	VAR jointtarget SDP_1960 := [[-7.34, 34.53, 8.17, 0, 47.31, -84.1], [9E9, 9E9, 9E9, 9E9, 9E9, 9E9]];
	VAR jointtarget SDP_1961 := [[-7.2, 34.54, 8.14, 0, 47.32, -83.96], [9E9, 9E9, 9E9, 9E9, 9E9, 9E9]];
	VAR jointtarget SDP_1962 := [[-7.06, 34.55, 8.12, 0, 47.33, -83.82], [9E9, 9E9, 9E9, 9E9, 9E9, 9E9]];
	VAR jointtarget SDP_1963 := [[-6.92, 34.57, 8.09, 0, 47.34, -83.68], [9E9, 9E9, 9E9, 9E9, 9E9, 9E9]];
	VAR jointtarget SDP_1964 := [[-6.79, 34.58, 8.06, 0, 47.36, -83.55], [9E9, 9E9, 9E9, 9E9, 9E9, 9E9]];
	VAR jointtarget SDP_1965 := [[-6.65, 34.6, 8.03, 0, 47.37, -83.41], [9E9, 9E9, 9E9, 9E9, 9E9, 9E9]];
	VAR jointtarget SDP_1966 := [[-6.51, 34.61, 8, 0, 47.38, -83.27], [9E9, 9E9, 9E9, 9E9, 9E9, 9E9]];
	VAR jointtarget SDP_1967 := [[-6.38, 34.63, 7.97, 0, 47.39, -83.14], [9E9, 9E9, 9E9, 9E9, 9E9, 9E9]];
	VAR jointtarget SDP_1968 := [[-6.24, 34.65, 7.94, 0, 47.41, -83], [9E9, 9E9, 9E9, 9E9, 9E9, 9E9]];
	VAR jointtarget SDP_1969 := [[-6.1, 34.66, 7.91, 0, 47.42, -82.86], [9E9, 9E9, 9E9, 9E9, 9E9, 9E9]];
	VAR jointtarget SDP_1970 := [[-6.07, 34.67, 7.91, 0, 47.43, -83.49], [9E9, 9E9, 9E9, 9E9, 9E9, 9E9]];
	VAR jointtarget SDP_1971 := [[-6.03, 34.67, 7.9, 0, 47.43, -84.78], [9E9, 9E9, 9E9, 9E9, 9E9, 9E9]];
	VAR jointtarget SDP_1972 := [[-6, 34.67, 7.9, 0, 47.43, -86.07], [9E9, 9E9, 9E9, 9E9, 9E9, 9E9]];
	VAR jointtarget SDP_1973 := [[-5.97, 34.67, 7.89, 0, 47.43, -87.36], [9E9, 9E9, 9E9, 9E9, 9E9, 9E9]];
	VAR jointtarget SDP_1974 := [[-5.93, 34.67, 7.89, 0, 47.43, -88.65], [9E9, 9E9, 9E9, 9E9, 9E9, 9E9]];
	VAR jointtarget SDP_1975 := [[-5.9, 34.67, 7.89, 0, 47.43, -89.94], [9E9, 9E9, 9E9, 9E9, 9E9, 9E9]];
	VAR jointtarget SDP_1976 := [[-5.86, 34.67, 7.89, 0, 47.43, -91.23], [9E9, 9E9, 9E9, 9E9, 9E9, 9E9]];
	VAR jointtarget SDP_1977 := [[-5.83, 34.67, 7.9, 0, 47.43, -92.52], [9E9, 9E9, 9E9, 9E9, 9E9, 9E9]];
	VAR jointtarget SDP_1978 := [[-5.79, 34.67, 7.9, 0, 47.43, -93.81], [9E9, 9E9, 9E9, 9E9, 9E9, 9E9]];
	VAR jointtarget SDP_1979 := [[-5.76, 34.67, 7.91, 0, 47.43, -95.1], [9E9, 9E9, 9E9, 9E9, 9E9, 9E9]];
	VAR jointtarget SDP_1980 := [[-4.6, 34.56, 8.1, 0, 47.35, -94.6], [9E9, 9E9, 9E9, 9E9, 9E9, 9E9]];
	VAR jointtarget SDP_1981 := [[-3.43, 34.47, 8.24, 0, 47.29, -93.43], [9E9, 9E9, 9E9, 9E9, 9E9, 9E9]];
	VAR jointtarget SDP_1982 := [[-2.26, 34.41, 8.34, 0, 47.25, -92.26], [9E9, 9E9, 9E9, 9E9, 9E9, 9E9]];
	VAR jointtarget SDP_1983 := [[-1.09, 34.37, 8.41, 0, 47.22, -91.09], [9E9, 9E9, 9E9, 9E9, 9E9, 9E9]];
	VAR jointtarget SDP_1984 := [[0.09, 34.36, 8.42, 0, 47.21, -89.91], [9E9, 9E9, 9E9, 9E9, 9E9, 9E9]];
	VAR jointtarget SDP_1985 := [[1.26, 34.38, 8.4, 0, 47.22, -88.74], [9E9, 9E9, 9E9, 9E9, 9E9, 9E9]];
	VAR jointtarget SDP_1986 := [[2.43, 34.42, 8.33, 0, 47.25, -87.57], [9E9, 9E9, 9E9, 9E9, 9E9, 9E9]];
	VAR jointtarget SDP_1987 := [[3.6, 34.48, 8.22, 0, 47.3, -86.4], [9E9, 9E9, 9E9, 9E9, 9E9, 9E9]];
	VAR jointtarget SDP_1988 := [[4.77, 34.57, 8.07, 0, 47.36, -85.23], [9E9, 9E9, 9E9, 9E9, 9E9, 9E9]];
	VAR jointtarget SDP_1989 := [[5.93, 34.68, 7.88, 0, 47.44, -84.07], [9E9, 9E9, 9E9, 9E9, 9E9, 9E9]];
	VAR jointtarget SDP_1990 := [[6.27, 34.75, 7.76, 0, 47.49, -79.23], [9E9, 9E9, 9E9, 9E9, 9E9, 9E9]];
	VAR jointtarget SDP_1991 := [[6.6, 34.88, 7.55, 0, 47.58, -69.9], [9E9, 9E9, 9E9, 9E9, 9E9, 9E9]];
	VAR jointtarget SDP_1992 := [[6.9, 35.06, 7.24, 0, 47.7, -60.6], [9E9, 9E9, 9E9, 9E9, 9E9, 9E9]];
	VAR jointtarget SDP_1993 := [[7.17, 35.29, 6.85, 0, 47.86, -51.33], [9E9, 9E9, 9E9, 9E9, 9E9, 9E9]];
	VAR jointtarget SDP_1994 := [[7.4, 35.56, 6.38, 0, 48.06, -42.1], [9E9, 9E9, 9E9, 9E9, 9E9, 9E9]];
	VAR jointtarget SDP_1995 := [[7.59, 35.87, 5.85, 0, 48.28, -32.91], [9E9, 9E9, 9E9, 9E9, 9E9, 9E9]];
	VAR jointtarget SDP_1996 := [[7.73, 36.21, 5.27, 0, 48.52, -23.77], [9E9, 9E9, 9E9, 9E9, 9E9, 9E9]];
	VAR jointtarget SDP_1997 := [[7.82, 36.57, 4.65, 0, 48.78, -14.68], [9E9, 9E9, 9E9, 9E9, 9E9, 9E9]];
	VAR jointtarget SDP_1998 := [[7.85, 36.94, 4.01, 0, 49.05, -5.65], [9E9, 9E9, 9E9, 9E9, 9E9, 9E9]];
	VAR jointtarget SDP_1999 := [[7.83, 37.32, 3.37, 0, 49.32, 3.33], [9E9, 9E9, 9E9, 9E9, 9E9, 9E9]];
	VAR jointtarget SDP_2000 := [[7.68, 38.57, 1.19, 0, 50.23, 7.68], [9E9, 9E9, 9E9, 9E9, 9E9, 9E9]];
	VAR jointtarget SDP_2001 := [[7.54, 39.84, -1.02, 0, 51.18, 7.54], [9E9, 9E9, 9E9, 9E9, 9E9, 9E9]];
	VAR jointtarget SDP_2002 := [[7.4, 41.13, -3.28, 0, 52.15, 7.4], [9E9, 9E9, 9E9, 9E9, 9E9, 9E9]];
	VAR jointtarget SDP_2003 := [[7.26, 42.45, -5.59, 0, 53.15, 7.26], [9E9, 9E9, 9E9, 9E9, 9E9, 9E9]];
	VAR jointtarget SDP_2004 := [[7.13, 43.78, -7.96, 0, 54.18, 7.13], [9E9, 9E9, 9E9, 9E9, 9E9, 9E9]];
	VAR jointtarget SDP_2005 := [[7.01, 45.14, -10.39, 0, 55.25, 7.01], [9E9, 9E9, 9E9, 9E9, 9E9, 9E9]];
	VAR jointtarget SDP_2006 := [[6.89, 46.54, -12.89, 0, 56.35, 6.89], [9E9, 9E9, 9E9, 9E9, 9E9, 9E9]];
	VAR jointtarget SDP_2007 := [[6.77, 47.96, -15.45, 0, 57.49, 6.77], [9E9, 9E9, 9E9, 9E9, 9E9, 9E9]];
	VAR jointtarget SDP_2008 := [[6.66, 49.43, -18.1, 0, 58.68, 6.66], [9E9, 9E9, 9E9, 9E9, 9E9, 9E9]];
	VAR jointtarget SDP_2009 := [[6.55, 50.94, -20.85, 0, 59.91, 6.55], [9E9, 9E9, 9E9, 9E9, 9E9, 9E9]];
	VAR jointtarget SDP_2010 := [[6.55, 50.98, -20.93, 0, 59.95, 5.89], [9E9, 9E9, 9E9, 9E9, 9E9, 9E9]];
	VAR jointtarget SDP_2011 := [[6.55, 51.03, -21.01, 0, 59.98, 4.56], [9E9, 9E9, 9E9, 9E9, 9E9, 9E9]];
	VAR jointtarget SDP_2012 := [[6.55, 51.07, -21.09, 0, 60.02, 3.24], [9E9, 9E9, 9E9, 9E9, 9E9, 9E9]];
	VAR jointtarget SDP_2013 := [[6.54, 51.12, -21.17, 0, 60.06, 1.91], [9E9, 9E9, 9E9, 9E9, 9E9, 9E9]];
	VAR jointtarget SDP_2014 := [[6.54, 51.16, -21.26, 0, 60.1, 0.59], [9E9, 9E9, 9E9, 9E9, 9E9, 9E9]];
	VAR jointtarget SDP_2015 := [[6.54, 51.21, -21.34, 0, 60.13, -0.74], [9E9, 9E9, 9E9, 9E9, 9E9, 9E9]];
	VAR jointtarget SDP_2016 := [[6.55, 51.25, -21.42, 0, 60.17, -2.06], [9E9, 9E9, 9E9, 9E9, 9E9, 9E9]];
	VAR jointtarget SDP_2017 := [[6.55, 51.3, -21.51, 0, 60.21, -3.38], [9E9, 9E9, 9E9, 9E9, 9E9, 9E9]];
	VAR jointtarget SDP_2018 := [[6.55, 51.34, -21.59, 0, 60.25, -4.7], [9E9, 9E9, 9E9, 9E9, 9E9, 9E9]];
	VAR jointtarget SDP_2019 := [[6.55, 51.39, -21.67, 0, 60.28, -6.03], [9E9, 9E9, 9E9, 9E9, 9E9, 9E9]];
	VAR jointtarget SDP_2020 := [[6.57, 51.57, -22.01, 0, 60.43, -6.68], [9E9, 9E9, 9E9, 9E9, 9E9, 9E9]];
	VAR jointtarget SDP_2021 := [[6.58, 51.76, -22.34, 0, 60.59, -6.66], [9E9, 9E9, 9E9, 9E9, 9E9, 9E9]];
	VAR jointtarget SDP_2022 := [[6.59, 51.94, -22.68, 0, 60.74, -6.65], [9E9, 9E9, 9E9, 9E9, 9E9, 9E9]];
	VAR jointtarget SDP_2023 := [[6.6, 52.13, -23.02, 0, 60.89, -6.64], [9E9, 9E9, 9E9, 9E9, 9E9, 9E9]];
	VAR jointtarget SDP_2024 := [[6.62, 52.31, -23.36, 0, 61.05, -6.62], [9E9, 9E9, 9E9, 9E9, 9E9, 9E9]];
	VAR jointtarget SDP_2025 := [[6.63, 52.5, -23.7, 0, 61.2, -6.61], [9E9, 9E9, 9E9, 9E9, 9E9, 9E9]];
	VAR jointtarget SDP_2026 := [[6.64, 52.69, -24.04, 0, 61.36, -6.6], [9E9, 9E9, 9E9, 9E9, 9E9, 9E9]];
	VAR jointtarget SDP_2027 := [[6.65, 52.87, -24.39, 0, 61.51, -6.59], [9E9, 9E9, 9E9, 9E9, 9E9, 9E9]];
	VAR jointtarget SDP_2028 := [[6.67, 53.06, -24.74, 0, 61.67, -6.57], [9E9, 9E9, 9E9, 9E9, 9E9, 9E9]];
	VAR jointtarget SDP_2029 := [[6.68, 53.25, -25.08, 0, 61.83, -6.56], [9E9, 9E9, 9E9, 9E9, 9E9, 9E9]];
	VAR jointtarget SDP_2030 := [[6.66, 53.63, -25.77, 0, 62.14, 3.75], [9E9, 9E9, 9E9, 9E9, 9E9, 9E9]];
	VAR jointtarget SDP_2031 := [[6.58, 53.97, -26.4, 0, 62.43, 24.31], [9E9, 9E9, 9E9, 9E9, 9E9, 9E9]];
	VAR jointtarget SDP_2032 := [[6.43, 54.24, -26.89, 0, 62.65, 44.81], [9E9, 9E9, 9E9, 9E9, 9E9, 9E9]];
	VAR jointtarget SDP_2033 := [[6.24, 54.4, -27.18, 0, 62.79, 65.27], [9E9, 9E9, 9E9, 9E9, 9E9, 9E9]];
	VAR jointtarget SDP_2034 := [[6.04, 54.43, -27.23, 0, 62.81, 85.71], [9E9, 9E9, 9E9, 9E9, 9E9, 9E9]];
	VAR jointtarget SDP_2035 := [[5.84, 54.32, -27.04, 0, 62.72, 106.16], [9E9, 9E9, 9E9, 9E9, 9E9, 9E9]];
	VAR jointtarget SDP_2036 := [[5.67, 54.09, -26.62, 0, 62.53, 126.64], [9E9, 9E9, 9E9, 9E9, 9E9, 9E9]];
	VAR jointtarget SDP_2037 := [[5.56, 53.77, -26.04, 0, 62.26, 147.18], [9E9, 9E9, 9E9, 9E9, 9E9, 9E9]];
	VAR jointtarget SDP_2038 := [[5.52, 53.41, -25.36, 0, 61.96, 167.78], [9E9, 9E9, 9E9, 9E9, 9E9, 9E9]];
	VAR jointtarget SDP_2039 := [[5.55, 53.04, -24.69, 0, 61.65, 188.46], [9E9, 9E9, 9E9, 9E9, 9E9, 9E9]];
	VAR jointtarget SDP_2040 := [[5.58, 52.86, -24.36, 0, 61.5, 198.82], [9E9, 9E9, 9E9, 9E9, 9E9, 9E9]];
	VAR jointtarget SDP_2041 := [[5.62, 52.68, -24.03, 0, 61.35, 198.86], [9E9, 9E9, 9E9, 9E9, 9E9, 9E9]];
	VAR jointtarget SDP_2042 := [[5.65, 52.5, -23.7, 0, 61.2, 198.89], [9E9, 9E9, 9E9, 9E9, 9E9, 9E9]];
	VAR jointtarget SDP_2043 := [[5.69, 52.32, -23.38, 0, 61.06, 198.93], [9E9, 9E9, 9E9, 9E9, 9E9, 9E9]];
	VAR jointtarget SDP_2044 := [[5.72, 52.15, -23.05, 0, 60.91, 198.96], [9E9, 9E9, 9E9, 9E9, 9E9, 9E9]];
	VAR jointtarget SDP_2045 := [[5.76, 51.97, -22.73, 0, 60.76, 199], [9E9, 9E9, 9E9, 9E9, 9E9, 9E9]];
	VAR jointtarget SDP_2046 := [[5.79, 51.79, -22.41, 0, 60.62, 199.03], [9E9, 9E9, 9E9, 9E9, 9E9, 9E9]];
	VAR jointtarget SDP_2047 := [[5.83, 51.62, -22.09, 0, 60.47, 199.07], [9E9, 9E9, 9E9, 9E9, 9E9, 9E9]];
	VAR jointtarget SDP_2048 := [[5.87, 51.44, -21.77, 0, 60.33, 199.11], [9E9, 9E9, 9E9, 9E9, 9E9, 9E9]];
	VAR jointtarget SDP_2049 := [[5.9, 51.27, -21.46, 0, 60.19, 199.14], [9E9, 9E9, 9E9, 9E9, 9E9, 9E9]];
	VAR jointtarget SDP_2050 := [[5.91, 51.23, -21.38, 0, 60.15, 198.49], [9E9, 9E9, 9E9, 9E9, 9E9, 9E9]];
	VAR jointtarget SDP_2051 := [[5.92, 51.18, -21.3, 0, 60.11, 197.17], [9E9, 9E9, 9E9, 9E9, 9E9, 9E9]];
	VAR jointtarget SDP_2052 := [[5.93, 51.14, -21.22, 0, 60.08, 195.86], [9E9, 9E9, 9E9, 9E9, 9E9, 9E9]];
	VAR jointtarget SDP_2053 := [[5.93, 51.1, -21.14, 0, 60.04, 194.54], [9E9, 9E9, 9E9, 9E9, 9E9, 9E9]];
	VAR jointtarget SDP_2054 := [[5.94, 51.05, -21.06, 0, 60.01, 193.22], [9E9, 9E9, 9E9, 9E9, 9E9, 9E9]];
	VAR jointtarget SDP_2055 := [[5.94, 51.01, -20.98, 0, 59.97, 191.9], [9E9, 9E9, 9E9, 9E9, 9E9, 9E9]];
	VAR jointtarget SDP_2056 := [[5.95, 50.96, -20.9, 0, 59.93, 190.58], [9E9, 9E9, 9E9, 9E9, 9E9, 9E9]];
	VAR jointtarget SDP_2057 := [[5.95, 50.92, -20.81, 0, 59.9, 189.26], [9E9, 9E9, 9E9, 9E9, 9E9, 9E9]];
	VAR jointtarget SDP_2058 := [[5.96, 50.87, -20.73, 0, 59.86, 187.94], [9E9, 9E9, 9E9, 9E9, 9E9, 9E9]];
	VAR jointtarget SDP_2059 := [[5.96, 50.83, -20.65, 0, 59.82, 186.62], [9E9, 9E9, 9E9, 9E9, 9E9, 9E9]];
	VAR jointtarget SDP_2060 := [[6.05, 49.42, -18.08, 0, 58.67, 186.05], [9E9, 9E9, 9E9, 9E9, 9E9, 9E9]];
	VAR jointtarget SDP_2061 := [[6.15, 48.04, -15.6, 0, 57.56, 186.15], [9E9, 9E9, 9E9, 9E9, 9E9, 9E9]];
	VAR jointtarget SDP_2062 := [[6.25, 46.7, -13.18, 0, 56.48, 186.25], [9E9, 9E9, 9E9, 9E9, 9E9, 9E9]];
	VAR jointtarget SDP_2063 := [[6.35, 45.39, -10.83, 0, 55.44, 186.35], [9E9, 9E9, 9E9, 9E9, 9E9, 9E9]];
	VAR jointtarget SDP_2064 := [[6.46, 44.11, -8.54, 0, 54.44, 186.46], [9E9, 9E9, 9E9, 9E9, 9E9, 9E9]];
	VAR jointtarget SDP_2065 := [[6.56, 42.85, -6.31, 0, 53.46, 186.56], [9E9, 9E9, 9E9, 9E9, 9E9, 9E9]];
	VAR jointtarget SDP_2066 := [[6.68, 41.61, -4.12, 0, 52.51, 186.68], [9E9, 9E9, 9E9, 9E9, 9E9, 9E9]];
	VAR jointtarget SDP_2067 := [[6.79, 40.39, -1.98, 0, 51.59, 186.79], [9E9, 9E9, 9E9, 9E9, 9E9, 9E9]];
	VAR jointtarget SDP_2068 := [[6.91, 39.19, 0.11, 0, 50.69, 186.91], [9E9, 9E9, 9E9, 9E9, 9E9, 9E9]];
	VAR jointtarget SDP_2069 := [[7.04, 38.01, 2.17, 0, 49.82, 187.04], [9E9, 9E9, 9E9, 9E9, 9E9, 9E9]];
	VAR jointtarget SDP_2070 := [[7.05, 37.63, 2.82, 0, 49.54, 182.55], [9E9, 9E9, 9E9, 9E9, 9E9, 9E9]];
	VAR jointtarget SDP_2071 := [[7.02, 37.26, 3.47, 0, 49.27, 173.52], [9E9, 9E9, 9E9, 9E9, 9E9, 9E9]];
	VAR jointtarget SDP_2072 := [[6.93, 36.9, 4.09, 0, 49.01, 164.43], [9E9, 9E9, 9E9, 9E9, 9E9, 9E9]];
	VAR jointtarget SDP_2073 := [[6.78, 36.56, 4.68, 0, 48.77, 155.28], [9E9, 9E9, 9E9, 9E9, 9E9, 9E9]];
	VAR jointtarget SDP_2074 := [[6.6, 36.25, 5.21, 0, 48.55, 146.1], [9E9, 9E9, 9E9, 9E9, 9E9, 9E9]];
	VAR jointtarget SDP_2075 := [[6.36, 35.98, 5.67, 0, 48.35, 136.86], [9E9, 9E9, 9E9, 9E9, 9E9, 9E9]];
	VAR jointtarget SDP_2076 := [[6.09, 35.75, 6.06, 0, 48.19, 127.59], [9E9, 9E9, 9E9, 9E9, 9E9, 9E9]];
	VAR jointtarget SDP_2077 := [[5.79, 35.57, 6.36, 0, 48.07, 118.29], [9E9, 9E9, 9E9, 9E9, 9E9, 9E9]];
	VAR jointtarget SDP_2078 := [[5.47, 35.45, 6.57, 0, 47.98, 108.97], [9E9, 9E9, 9E9, 9E9, 9E9, 9E9]];
	VAR jointtarget SDP_2079 := [[5.13, 35.39, 6.68, 0, 47.93, 99.63], [9E9, 9E9, 9E9, 9E9, 9E9, 9E9]];
	VAR jointtarget SDP_2080 := [[4.07, 35.3, 6.83, 0, 47.87, 94.07], [9E9, 9E9, 9E9, 9E9, 9E9, 9E9]];
	VAR jointtarget SDP_2081 := [[3.01, 35.23, 6.95, 0, 47.82, 93.01], [9E9, 9E9, 9E9, 9E9, 9E9, 9E9]];
	VAR jointtarget SDP_2082 := [[1.95, 35.18, 7.04, 0, 47.79, 91.95], [9E9, 9E9, 9E9, 9E9, 9E9, 9E9]];
	VAR jointtarget SDP_2083 := [[0.89, 35.15, 7.08, 0, 47.77, 90.89], [9E9, 9E9, 9E9, 9E9, 9E9, 9E9]];
	VAR jointtarget SDP_2084 := [[-0.18, 35.14, 7.1, 0, 47.76, 89.82], [9E9, 9E9, 9E9, 9E9, 9E9, 9E9]];
	VAR jointtarget SDP_2085 := [[-1.24, 35.16, 7.07, 0, 47.77, 88.76], [9E9, 9E9, 9E9, 9E9, 9E9, 9E9]];
	VAR jointtarget SDP_2086 := [[-2.31, 35.19, 7.01, 0, 47.8, 87.69], [9E9, 9E9, 9E9, 9E9, 9E9, 9E9]];
	VAR jointtarget SDP_2087 := [[-3.37, 35.25, 6.92, 0, 47.84, 86.63], [9E9, 9E9, 9E9, 9E9, 9E9, 9E9]];
	VAR jointtarget SDP_2088 := [[-4.43, 35.33, 6.78, 0, 47.89, 85.57], [9E9, 9E9, 9E9, 9E9, 9E9, 9E9]];
	VAR jointtarget SDP_2089 := [[-5.48, 35.42, 6.62, 0, 47.96, 84.52], [9E9, 9E9, 9E9, 9E9, 9E9, 9E9]];
	VAR jointtarget SDP_2090 := [[-5.59, 35.43, 6.6, 0, 47.96, 86.6], [9E9, 9E9, 9E9, 9E9, 9E9, 9E9]];
	VAR jointtarget SDP_2091 := [[-5.71, 35.43, 6.61, 0, 47.96, 90.88], [9E9, 9E9, 9E9, 9E9, 9E9, 9E9]];
	VAR jointtarget SDP_2092 := [[-5.82, 35.42, 6.63, 0, 47.96, 95.15], [9E9, 9E9, 9E9, 9E9, 9E9, 9E9]];
	VAR jointtarget SDP_2093 := [[-5.93, 35.4, 6.66, 0, 47.94, 99.43], [9E9, 9E9, 9E9, 9E9, 9E9, 9E9]];
	VAR jointtarget SDP_2094 := [[-6.04, 35.37, 6.71, 0, 47.92, 103.71], [9E9, 9E9, 9E9, 9E9, 9E9, 9E9]];
	VAR jointtarget SDP_2095 := [[-6.14, 35.33, 6.77, 0, 47.9, 107.99], [9E9, 9E9, 9E9, 9E9, 9E9, 9E9]];
	VAR jointtarget SDP_2096 := [[-6.25, 35.29, 6.85, 0, 47.86, 112.27], [9E9, 9E9, 9E9, 9E9, 9E9, 9E9]];
	VAR jointtarget SDP_2097 := [[-6.35, 35.23, 6.94, 0, 47.83, 116.56], [9E9, 9E9, 9E9, 9E9, 9E9, 9E9]];
	VAR jointtarget SDP_2098 := [[-6.44, 35.17, 7.05, 0, 47.78, 120.85], [9E9, 9E9, 9E9, 9E9, 9E9, 9E9]];
	VAR jointtarget SDP_2099 := [[-6.54, 35.1, 7.16, 0, 47.73, 125.15], [9E9, 9E9, 9E9, 9E9, 9E9, 9E9]];
	VAR jointtarget SDP_2100 := [[-6.59, 35.06, 7.24, 0, 47.7, 127.29], [9E9, 9E9, 9E9, 9E9, 9E9, 9E9]];
	VAR jointtarget SDP_2101 := [[-6.64, 35.01, 7.31, 0, 47.67, 127.23], [9E9, 9E9, 9E9, 9E9, 9E9, 9E9]];
	VAR jointtarget SDP_2102 := [[-6.7, 34.97, 7.39, 0, 47.64, 127.18], [9E9, 9E9, 9E9, 9E9, 9E9, 9E9]];
	VAR jointtarget SDP_2103 := [[-6.75, 34.93, 7.46, 0, 47.61, 127.12], [9E9, 9E9, 9E9, 9E9, 9E9, 9E9]];
	VAR jointtarget SDP_2104 := [[-6.81, 34.88, 7.54, 0, 47.58, 127.07], [9E9, 9E9, 9E9, 9E9, 9E9, 9E9]];
	VAR jointtarget SDP_2105 := [[-6.86, 34.84, 7.61, 0, 47.55, 127.01], [9E9, 9E9, 9E9, 9E9, 9E9, 9E9]];
	VAR jointtarget SDP_2106 := [[-6.92, 34.8, 7.69, 0, 47.52, 126.96], [9E9, 9E9, 9E9, 9E9, 9E9, 9E9]];
	VAR jointtarget SDP_2107 := [[-6.97, 34.75, 7.76, 0, 47.49, 126.91], [9E9, 9E9, 9E9, 9E9, 9E9, 9E9]];
	VAR jointtarget SDP_2108 := [[-7.03, 34.71, 7.83, 0, 47.46, 126.85], [9E9, 9E9, 9E9, 9E9, 9E9, 9E9]];
	VAR jointtarget SDP_2109 := [[-7.08, 34.67, 7.91, 0, 47.43, 126.8], [9E9, 9E9, 9E9, 9E9, 9E9, 9E9]];
	VAR jointtarget SDP_2110 := [[-7.39, 34.53, 8.14, 0, 47.33, 113.1], [9E9, 9E9, 9E9, 9E9, 9E9, 9E9]];
	VAR jointtarget SDP_2111 := [[-7.72, 34.55, 8.1, 0, 47.35, 85.99], [9E9, 9E9, 9E9, 9E9, 9E9, 9E9]];
	VAR jointtarget SDP_2112 := [[-8.01, 34.73, 7.8, 0, 47.47, 58.93], [9E9, 9E9, 9E9, 9E9, 9E9, 9E9]];
	VAR jointtarget SDP_2113 := [[-8.18, 35.03, 7.29, 0, 47.68, 31.98], [9E9, 9E9, 9E9, 9E9, 9E9, 9E9]];
	VAR jointtarget SDP_2114 := [[-8.21, 35.38, 6.69, 0, 47.93, 5.18], [9E9, 9E9, 9E9, 9E9, 9E9, 9E9]];
	VAR jointtarget SDP_2115 := [[-8.09, 35.71, 6.13, 0, 48.16, -21.48], [9E9, 9E9, 9E9, 9E9, 9E9, 9E9]];
	VAR jointtarget SDP_2116 := [[-7.85, 35.95, 5.73, 0, 48.33, -48.01], [9E9, 9E9, 9E9, 9E9, 9E9, 9E9]];
	VAR jointtarget SDP_2117 := [[-7.53, 36.04, 5.56, 0, 48.4, -74.47], [9E9, 9E9, 9E9, 9E9, 9E9, 9E9]];
	VAR jointtarget SDP_2118 := [[-7.21, 35.97, 5.68, 0, 48.35, -100.93], [9E9, 9E9, 9E9, 9E9, 9E9, 9E9]];
	VAR jointtarget SDP_2119 := [[-6.96, 35.75, 6.05, 0, 48.19, -127.44], [9E9, 9E9, 9E9, 9E9, 9E9, 9E9]];
	VAR jointtarget SDP_2120 := [[-6.9, 35.68, 6.17, 0, 48.14, -140.78], [9E9, 9E9, 9E9, 9E9, 9E9, 9E9]];
	VAR jointtarget SDP_2121 := [[-6.85, 35.61, 6.3, 0, 48.09, -140.72], [9E9, 9E9, 9E9, 9E9, 9E9, 9E9]];
	VAR jointtarget SDP_2122 := [[-6.79, 35.54, 6.42, 0, 48.04, -140.67], [9E9, 9E9, 9E9, 9E9, 9E9, 9E9]];
	VAR jointtarget SDP_2123 := [[-6.74, 35.47, 6.54, 0, 47.99, -140.62], [9E9, 9E9, 9E9, 9E9, 9E9, 9E9]];
	VAR jointtarget SDP_2124 := [[-6.68, 35.4, 6.66, 0, 47.94, -140.56], [9E9, 9E9, 9E9, 9E9, 9E9, 9E9]];
	VAR jointtarget SDP_2125 := [[-6.63, 35.33, 6.78, 0, 47.89, -140.51], [9E9, 9E9, 9E9, 9E9, 9E9, 9E9]];
	VAR jointtarget SDP_2126 := [[-6.58, 35.26, 6.9, 0, 47.84, -140.45], [9E9, 9E9, 9E9, 9E9, 9E9, 9E9]];
	VAR jointtarget SDP_2127 := [[-6.52, 35.19, 7.02, 0, 47.79, -140.4], [9E9, 9E9, 9E9, 9E9, 9E9, 9E9]];
	VAR jointtarget SDP_2128 := [[-6.47, 35.11, 7.14, 0, 47.74, -140.34], [9E9, 9E9, 9E9, 9E9, 9E9, 9E9]];
	VAR jointtarget SDP_2129 := [[-6.41, 35.04, 7.26, 0, 47.69, -140.29], [9E9, 9E9, 9E9, 9E9, 9E9, 9E9]];
	VAR jointtarget SDP_2130 := [[-6.38, 35.01, 7.32, 0, 47.67, -139.16], [9E9, 9E9, 9E9, 9E9, 9E9, 9E9]];
	VAR jointtarget SDP_2131 := [[-6.36, 34.98, 7.37, 0, 47.65, -136.92], [9E9, 9E9, 9E9, 9E9, 9E9, 9E9]];
	VAR jointtarget SDP_2132 := [[-6.33, 34.95, 7.42, 0, 47.63, -134.69], [9E9, 9E9, 9E9, 9E9, 9E9, 9E9]];
	VAR jointtarget SDP_2133 := [[-6.3, 34.92, 7.47, 0, 47.61, -132.45], [9E9, 9E9, 9E9, 9E9, 9E9, 9E9]];
	VAR jointtarget SDP_2134 := [[-6.27, 34.9, 7.51, 0, 47.59, -130.22], [9E9, 9E9, 9E9, 9E9, 9E9, 9E9]];
	VAR jointtarget SDP_2135 := [[-6.24, 34.87, 7.56, 0, 47.57, -127.98], [9E9, 9E9, 9E9, 9E9, 9E9, 9E9]];
	VAR jointtarget SDP_2136 := [[-6.21, 34.84, 7.6, 0, 47.56, -125.74], [9E9, 9E9, 9E9, 9E9, 9E9, 9E9]];
	VAR jointtarget SDP_2137 := [[-6.18, 34.82, 7.64, 0, 47.54, -123.5], [9E9, 9E9, 9E9, 9E9, 9E9, 9E9]];
	VAR jointtarget SDP_2138 := [[-6.14, 34.8, 7.67, 0, 47.53, -121.26], [9E9, 9E9, 9E9, 9E9, 9E9, 9E9]];
	VAR jointtarget SDP_2139 := [[-6.11, 34.78, 7.71, 0, 47.52, -119.01], [9E9, 9E9, 9E9, 9E9, 9E9, 9E9]];
	VAR jointtarget SDP_2140 := [[-6.09, 34.77, 7.72, 0, 47.51, -117.89], [9E9, 9E9, 9E9, 9E9, 9E9, 9E9]];
	VAR jointtarget SDP_2141 := [[-6.07, 34.76, 7.74, 0, 47.5, -117.87], [9E9, 9E9, 9E9, 9E9, 9E9, 9E9]];
	VAR jointtarget SDP_2142 := [[-6.05, 34.74, 7.76, 0, 47.5, -117.86], [9E9, 9E9, 9E9, 9E9, 9E9, 9E9]];
	VAR jointtarget SDP_2143 := [[-6.04, 34.73, 7.77, 0, 47.49, -117.84], [9E9, 9E9, 9E9, 9E9, 9E9, 9E9]];
	VAR jointtarget SDP_2144 := [[-6.02, 34.72, 7.79, 0, 47.49, -117.82], [9E9, 9E9, 9E9, 9E9, 9E9, 9E9]];
	VAR jointtarget SDP_2145 := [[-6, 34.71, 7.81, 0, 47.48, -117.8], [9E9, 9E9, 9E9, 9E9, 9E9, 9E9]];
	VAR jointtarget SDP_2146 := [[-5.98, 34.7, 7.82, 0, 47.47, -117.79], [9E9, 9E9, 9E9, 9E9, 9E9, 9E9]];
	VAR jointtarget SDP_2147 := [[-5.97, 34.69, 7.84, 0, 47.47, -117.77], [9E9, 9E9, 9E9, 9E9, 9E9, 9E9]];
	VAR jointtarget SDP_2148 := [[-5.95, 34.68, 7.86, 0, 47.46, -117.75], [9E9, 9E9, 9E9, 9E9, 9E9, 9E9]];
	VAR jointtarget SDP_2149 := [[-5.93, 34.67, 7.87, 0, 47.46, -117.73], [9E9, 9E9, 9E9, 9E9, 9E9, 9E9]];
	VAR jointtarget SDP_2150 := [[-4.75, 34.56, 8.07, 0, 47.37, -94.75], [9E9, 9E9, 9E9, 9E9, 9E9, 9E9]];
	VAR jointtarget SDP_2151 := [[-3.57, 34.46, 8.22, 0, 47.31, -93.57], [9E9, 9E9, 9E9, 9E9, 9E9, 9E9]];
	VAR jointtarget SDP_2152 := [[-2.38, 34.4, 8.33, 0, 47.27, -92.38], [9E9, 9E9, 9E9, 9E9, 9E9, 9E9]];
	VAR jointtarget SDP_2153 := [[-1.19, 34.36, 8.4, 0, 47.24, -91.19], [9E9, 9E9, 9E9, 9E9, 9E9, 9E9]];
	VAR jointtarget SDP_2154 := [[0, 34.35, 8.42, 0, 47.23, -90], [9E9, 9E9, 9E9, 9E9, 9E9, 9E9]];
	VAR jointtarget SDP_2155 := [[1.19, 34.36, 8.4, 0, 47.24, -88.81], [9E9, 9E9, 9E9, 9E9, 9E9, 9E9]];
	VAR jointtarget SDP_2156 := [[2.38, 34.4, 8.33, 0, 47.27, -87.62], [9E9, 9E9, 9E9, 9E9, 9E9, 9E9]];
	VAR jointtarget SDP_2157 := [[3.57, 34.46, 8.22, 0, 47.31, -86.43], [9E9, 9E9, 9E9, 9E9, 9E9, 9E9]];
	VAR jointtarget SDP_2158 := [[4.75, 34.56, 8.07, 0, 47.37, -85.25], [9E9, 9E9, 9E9, 9E9, 9E9, 9E9]];
	VAR jointtarget SDP_2159 := [[5.93, 34.67, 7.87, 0, 47.46, -84.07], [9E9, 9E9, 9E9, 9E9, 9E9, 9E9]];
	VAR jointtarget SDP_2160 := [[6.27, 34.74, 7.76, 0, 47.5, -79.23], [9E9, 9E9, 9E9, 9E9, 9E9, 9E9]];
	VAR jointtarget SDP_2161 := [[6.6, 34.86, 7.54, 0, 47.59, -69.9], [9E9, 9E9, 9E9, 9E9, 9E9, 9E9]];
	VAR jointtarget SDP_2162 := [[6.9, 35.04, 7.24, 0, 47.72, -60.6], [9E9, 9E9, 9E9, 9E9, 9E9, 9E9]];
	VAR jointtarget SDP_2163 := [[7.17, 35.27, 6.85, 0, 47.88, -51.33], [9E9, 9E9, 9E9, 9E9, 9E9, 9E9]];
	VAR jointtarget SDP_2164 := [[7.4, 35.55, 6.38, 0, 48.07, -42.1], [9E9, 9E9, 9E9, 9E9, 9E9, 9E9]];
	VAR jointtarget SDP_2165 := [[7.59, 35.86, 5.85, 0, 48.29, -32.91], [9E9, 9E9, 9E9, 9E9, 9E9, 9E9]];
	VAR jointtarget SDP_2166 := [[7.73, 36.2, 5.27, 0, 48.54, -23.77], [9E9, 9E9, 9E9, 9E9, 9E9, 9E9]];
	VAR jointtarget SDP_2167 := [[7.82, 36.56, 4.65, 0, 48.79, -14.68], [9E9, 9E9, 9E9, 9E9, 9E9, 9E9]];
	VAR jointtarget SDP_2168 := [[7.85, 36.93, 4.01, 0, 49.06, -5.65], [9E9, 9E9, 9E9, 9E9, 9E9, 9E9]];
	VAR jointtarget SDP_2169 := [[7.83, 37.31, 3.36, 0, 49.33, 3.33], [9E9, 9E9, 9E9, 9E9, 9E9, 9E9]];
	VAR jointtarget SDP_2170 := [[7.68, 38.54, 1.23, 0, 50.23, 7.68], [9E9, 9E9, 9E9, 9E9, 9E9, 9E9]];
	VAR jointtarget SDP_2171 := [[7.54, 39.79, -0.94, 0, 51.16, 7.54], [9E9, 9E9, 9E9, 9E9, 9E9, 9E9]];
	VAR jointtarget SDP_2172 := [[7.4, 41.05, -3.16, 0, 52.11, 7.4], [9E9, 9E9, 9E9, 9E9, 9E9, 9E9]];
	VAR jointtarget SDP_2173 := [[7.27, 42.34, -5.43, 0, 53.09, 7.27], [9E9, 9E9, 9E9, 9E9, 9E9, 9E9]];
	VAR jointtarget SDP_2174 := [[7.15, 43.65, -7.75, 0, 54.1, 7.15], [9E9, 9E9, 9E9, 9E9, 9E9, 9E9]];
	VAR jointtarget SDP_2175 := [[7.02, 44.98, -10.13, 0, 55.15, 7.02], [9E9, 9E9, 9E9, 9E9, 9E9, 9E9]];
	VAR jointtarget SDP_2176 := [[6.9, 46.35, -12.57, 0, 56.22, 6.9], [9E9, 9E9, 9E9, 9E9, 9E9, 9E9]];
	VAR jointtarget SDP_2177 := [[6.79, 47.75, -15.09, 0, 57.34, 6.79], [9E9, 9E9, 9E9, 9E9, 9E9, 9E9]];
	VAR jointtarget SDP_2178 := [[6.68, 49.18, -17.68, 0, 58.5, 6.68], [9E9, 9E9, 9E9, 9E9, 9E9, 9E9]];
	VAR jointtarget SDP_2179 := [[6.57, 50.65, -20.35, 0, 59.7, 6.57], [9E9, 9E9, 9E9, 9E9, 9E9, 9E9]];
	VAR jointtarget SDP_2180 := [[6.56, 50.8, -20.62, 0, 59.82, 8.75], [9E9, 9E9, 9E9, 9E9, 9E9, 9E9]];
	VAR jointtarget SDP_2181 := [[6.54, 50.95, -20.89, 0, 59.94, 13.12], [9E9, 9E9, 9E9, 9E9, 9E9, 9E9]];
	VAR jointtarget SDP_2182 := [[6.51, 51.09, -21.15, 0, 60.06, 17.48], [9E9, 9E9, 9E9, 9E9, 9E9, 9E9]];
	VAR jointtarget SDP_2183 := [[6.48, 51.23, -21.4, 0, 60.17, 21.83], [9E9, 9E9, 9E9, 9E9, 9E9, 9E9]];
	VAR jointtarget SDP_2184 := [[6.44, 51.36, -21.65, 0, 60.28, 26.18], [9E9, 9E9, 9E9, 9E9, 9E9, 9E9]];
	VAR jointtarget SDP_2185 := [[6.39, 51.49, -21.89, 0, 60.39, 30.52], [9E9, 9E9, 9E9, 9E9, 9E9, 9E9]];
	VAR jointtarget SDP_2186 := [[6.34, 51.62, -22.11, 0, 60.49, 34.86], [9E9, 9E9, 9E9, 9E9, 9E9, 9E9]];
	VAR jointtarget SDP_2187 := [[6.28, 51.74, -22.33, 0, 60.59, 39.19], [9E9, 9E9, 9E9, 9E9, 9E9, 9E9]];
	VAR jointtarget SDP_2188 := [[6.22, 51.85, -22.53, 0, 60.68, 43.51], [9E9, 9E9, 9E9, 9E9, 9E9, 9E9]];
	VAR jointtarget SDP_2189 := [[6.15, 51.95, -22.72, 0, 60.77, 47.83], [9E9, 9E9, 9E9, 9E9, 9E9, 9E9]];
	VAR jointtarget SDP_2190 := [[6.11, 52.01, -22.83, 0, 60.82, 49.99], [9E9, 9E9, 9E9, 9E9, 9E9, 9E9]];
	VAR jointtarget SDP_2191 := [[6.07, 52.07, -22.94, 0, 60.87, 49.95], [9E9, 9E9, 9E9, 9E9, 9E9, 9E9]];
	VAR jointtarget SDP_2192 := [[6.03, 52.13, -23.04, 0, 60.92, 49.9], [9E9, 9E9, 9E9, 9E9, 9E9, 9E9]];
	VAR jointtarget SDP_2193 := [[5.99, 52.19, -23.15, 0, 60.97, 49.86], [9E9, 9E9, 9E9, 9E9, 9E9, 9E9]];
	VAR jointtarget SDP_2194 := [[5.94, 52.25, -23.26, 0, 61.02, 49.82], [9E9, 9E9, 9E9, 9E9, 9E9, 9E9]];
	VAR jointtarget SDP_2195 := [[5.9, 52.31, -23.37, 0, 61.06, 49.78], [9E9, 9E9, 9E9, 9E9, 9E9, 9E9]];
	VAR jointtarget SDP_2196 := [[5.86, 52.37, -23.48, 0, 61.11, 49.74], [9E9, 9E9, 9E9, 9E9, 9E9, 9E9]];
	VAR jointtarget SDP_2197 := [[5.82, 52.43, -23.59, 0, 61.17, 49.7], [9E9, 9E9, 9E9, 9E9, 9E9, 9E9]];
	VAR jointtarget SDP_2198 := [[5.78, 52.49, -23.71, 0, 61.22, 49.66], [9E9, 9E9, 9E9, 9E9, 9E9, 9E9]];
	VAR jointtarget SDP_2199 := [[5.74, 52.55, -23.82, 0, 61.27, 49.61], [9E9, 9E9, 9E9, 9E9, 9E9, 9E9]];
	VAR jointtarget SDP_2200 := [[5.58, 52.92, -24.49, 0, 61.57, 36.07], [9E9, 9E9, 9E9, 9E9, 9E9, 9E9]];
	VAR jointtarget SDP_2201 := [[5.54, 53.38, -25.33, 0, 61.95, 9.25], [9E9, 9E9, 9E9, 9E9, 9E9, 9E9]];
	VAR jointtarget SDP_2202 := [[5.62, 53.82, -26.15, 0, 62.32, -17.44], [9E9, 9E9, 9E9, 9E9, 9E9, 9E9]];
	VAR jointtarget SDP_2203 := [[5.8, 54.16, -26.77, 0, 62.61, -44.04], [9E9, 9E9, 9E9, 9E9, 9E9, 9E9]];
	VAR jointtarget SDP_2204 := [[6.04, 54.32, -27.06, 0, 62.74, -70.57], [9E9, 9E9, 9E9, 9E9, 9E9, 9E9]];
	VAR jointtarget SDP_2205 := [[6.3, 54.26, -26.95, 0, 62.69, -97.09], [9E9, 9E9, 9E9, 9E9, 9E9, 9E9]];
	VAR jointtarget SDP_2206 := [[6.51, 53.99, -26.46, 0, 62.47, -123.65], [9E9, 9E9, 9E9, 9E9, 9E9, 9E9]];
	VAR jointtarget SDP_2207 := [[6.64, 53.59, -25.72, 0, 62.13, -150.3], [9E9, 9E9, 9E9, 9E9, 9E9, 9E9]];
	VAR jointtarget SDP_2208 := [[6.66, 53.12, -24.86, 0, 61.74, -177.06], [9E9, 9E9, 9E9, 9E9, 9E9, 9E9]];
	VAR jointtarget SDP_2209 := [[6.55, 52.7, -24.1, 0, 61.39, -203.94], [9E9, 9E9, 9E9, 9E9, 9E9, 9E9]];
	VAR jointtarget SDP_2210 := [[6.52, 52.63, -23.96, 0, 61.33, -217.36], [9E9, 9E9, 9E9, 9E9, 9E9, 9E9]];
	VAR jointtarget SDP_2211 := [[6.48, 52.55, -23.82, 0, 61.27, -217.39], [9E9, 9E9, 9E9, 9E9, 9E9, 9E9]];
	VAR jointtarget SDP_2212 := [[6.45, 52.48, -23.69, 0, 61.21, -217.42], [9E9, 9E9, 9E9, 9E9, 9E9, 9E9]];
	VAR jointtarget SDP_2213 := [[6.42, 52.4, -23.55, 0, 61.14, -217.46], [9E9, 9E9, 9E9, 9E9, 9E9, 9E9]];
	VAR jointtarget SDP_2214 := [[6.39, 52.33, -23.41, 0, 61.08, -217.49], [9E9, 9E9, 9E9, 9E9, 9E9, 9E9]];
	VAR jointtarget SDP_2215 := [[6.35, 52.26, -23.28, 0, 61.02, -217.52], [9E9, 9E9, 9E9, 9E9, 9E9, 9E9]];
	VAR jointtarget SDP_2216 := [[6.32, 52.18, -23.14, 0, 60.96, -217.56], [9E9, 9E9, 9E9, 9E9, 9E9, 9E9]];
	VAR jointtarget SDP_2217 := [[6.29, 52.11, -23.01, 0, 60.9, -217.59], [9E9, 9E9, 9E9, 9E9, 9E9, 9E9]];
	VAR jointtarget SDP_2218 := [[6.25, 52.04, -22.87, 0, 60.84, -217.62], [9E9, 9E9, 9E9, 9E9, 9E9, 9E9]];
	VAR jointtarget SDP_2219 := [[6.22, 51.96, -22.74, 0, 60.78, -217.66], [9E9, 9E9, 9E9, 9E9, 9E9, 9E9]];
	VAR jointtarget SDP_2220 := [[6.17, 51.84, -22.51, 0, 60.68, -215.51], [9E9, 9E9, 9E9, 9E9, 9E9, 9E9]];
	VAR jointtarget SDP_2221 := [[6.12, 51.71, -22.27, 0, 60.57, -211.17], [9E9, 9E9, 9E9, 9E9, 9E9, 9E9]];
	VAR jointtarget SDP_2222 := [[6.08, 51.57, -22.03, 0, 60.46, -206.83], [9E9, 9E9, 9E9, 9E9, 9E9, 9E9]];
	VAR jointtarget SDP_2223 := [[6.05, 51.43, -21.77, 0, 60.34, -202.47], [9E9, 9E9, 9E9, 9E9, 9E9, 9E9]];
	VAR jointtarget SDP_2224 := [[6.02, 51.29, -21.51, 0, 60.22, -198.11], [9E9, 9E9, 9E9, 9E9, 9E9, 9E9]];
	VAR jointtarget SDP_2225 := [[6, 51.14, -21.24, 0, 60.1, -193.75], [9E9, 9E9, 9E9, 9E9, 9E9, 9E9]];
	VAR jointtarget SDP_2226 := [[5.98, 50.99, -20.97, 0, 59.98, -189.38], [9E9, 9E9, 9E9, 9E9, 9E9, 9E9]];
	VAR jointtarget SDP_2227 := [[5.97, 50.84, -20.7, 0, 59.86, -185], [9E9, 9E9, 9E9, 9E9, 9E9, 9E9]];
	VAR jointtarget SDP_2228 := [[5.97, 50.69, -20.43, 0, 59.73, -180.61], [9E9, 9E9, 9E9, 9E9, 9E9, 9E9]];
	VAR jointtarget SDP_2229 := [[5.98, 50.55, -20.16, 0, 59.61, -176.22], [9E9, 9E9, 9E9, 9E9, 9E9, 9E9]];
	VAR jointtarget SDP_2230 := [[6.07, 49.17, -17.66, 0, 58.49, -173.93], [9E9, 9E9, 9E9, 9E9, 9E9, 9E9]];
	VAR jointtarget SDP_2231 := [[6.16, 47.82, -15.23, 0, 57.4, -173.84], [9E9, 9E9, 9E9, 9E9, 9E9, 9E9]];
	VAR jointtarget SDP_2232 := [[6.26, 46.51, -12.87, 0, 56.35, -173.74], [9E9, 9E9, 9E9, 9E9, 9E9, 9E9]];
	VAR jointtarget SDP_2233 := [[6.36, 45.23, -10.57, 0, 55.34, -173.64], [9E9, 9E9, 9E9, 9E9, 9E9, 9E9]];
	VAR jointtarget SDP_2234 := [[6.47, 43.98, -8.33, 0, 54.36, -173.53], [9E9, 9E9, 9E9, 9E9, 9E9, 9E9]];
	VAR jointtarget SDP_2235 := [[6.57, 42.74, -6.14, 0, 53.4, -173.43], [9E9, 9E9, 9E9, 9E9, 9E9, 9E9]];
	VAR jointtarget SDP_2236 := [[6.68, 41.53, -4, 0, 52.47, -173.32], [9E9, 9E9, 9E9, 9E9, 9E9, 9E9]];
	VAR jointtarget SDP_2237 := [[6.8, 40.34, -1.9, 0, 51.57, -173.2], [9E9, 9E9, 9E9, 9E9, 9E9, 9E9]];
	VAR jointtarget SDP_2238 := [[6.92, 39.16, 0.15, 0, 50.69, -173.08], [9E9, 9E9, 9E9, 9E9, 9E9, 9E9]];
	VAR jointtarget SDP_2239 := [[7.04, 38, 2.17, 0, 49.83, -172.96], [9E9, 9E9, 9E9, 9E9, 9E9, 9E9]];
	VAR jointtarget SDP_2240 := [[7.05, 37.62, 2.82, 0, 49.56, -177.45], [9E9, 9E9, 9E9, 9E9, 9E9, 9E9]];
	VAR jointtarget SDP_2241 := [[7.02, 37.24, 3.47, 0, 49.29, -186.48], [9E9, 9E9, 9E9, 9E9, 9E9, 9E9]];
	VAR jointtarget SDP_2242 := [[6.93, 36.88, 4.09, 0, 49.03, -195.57], [9E9, 9E9, 9E9, 9E9, 9E9, 9E9]];
	VAR jointtarget SDP_2243 := [[6.78, 36.54, 4.67, 0, 48.78, -204.72], [9E9, 9E9, 9E9, 9E9, 9E9, 9E9]];
	VAR jointtarget SDP_2244 := [[6.6, 36.23, 5.2, 0, 48.56, -213.9], [9E9, 9E9, 9E9, 9E9, 9E9, 9E9]];
	VAR jointtarget SDP_2245 := [[6.36, 35.96, 5.67, 0, 48.37, -223.14], [9E9, 9E9, 9E9, 9E9, 9E9, 9E9]];
	VAR jointtarget SDP_2246 := [[6.09, 35.74, 6.06, 0, 48.21, -232.41], [9E9, 9E9, 9E9, 9E9, 9E9, 9E9]];
	VAR jointtarget SDP_2247 := [[5.79, 35.56, 6.36, 0, 48.08, -241.71], [9E9, 9E9, 9E9, 9E9, 9E9, 9E9]];
	VAR jointtarget SDP_2248 := [[5.47, 35.44, 6.57, 0, 47.99, -251.03], [9E9, 9E9, 9E9, 9E9, 9E9, 9E9]];
	VAR jointtarget SDP_2249 := [[5.13, 35.38, 6.67, 0, 47.95, -260.37], [9E9, 9E9, 9E9, 9E9, 9E9, 9E9]];
	VAR jointtarget SDP_2250 := [[4.05, 35.28, 6.83, 0, 47.89, -265.95], [9E9, 9E9, 9E9, 9E9, 9E9, 9E9]];
	VAR jointtarget SDP_2251 := [[2.97, 35.21, 6.95, 0, 47.84, -267.03], [9E9, 9E9, 9E9, 9E9, 9E9, 9E9]];
	VAR jointtarget SDP_2252 := [[1.89, 35.16, 7.04, 0, 47.8, -268.11], [9E9, 9E9, 9E9, 9E9, 9E9, 9E9]];
	VAR jointtarget SDP_2253 := [[0.8, 35.14, 7.08, 0, 47.78, -269.2], [9E9, 9E9, 9E9, 9E9, 9E9, 9E9]];
	VAR jointtarget SDP_2254 := [[-0.28, 35.13, 7.09, 0, 47.78, -270.28], [9E9, 9E9, 9E9, 9E9, 9E9, 9E9]];
	VAR jointtarget SDP_2255 := [[-1.37, 35.15, 7.06, 0, 47.79, -271.37], [9E9, 9E9, 9E9, 9E9, 9E9, 9E9]];
	VAR jointtarget SDP_2256 := [[-2.45, 35.19, 7, 0, 47.82, -272.45], [9E9, 9E9, 9E9, 9E9, 9E9, 9E9]];
	VAR jointtarget SDP_2257 := [[-3.53, 35.25, 6.9, 0, 47.86, -273.53], [9E9, 9E9, 9E9, 9E9, 9E9, 9E9]];
	VAR jointtarget SDP_2258 := [[-4.61, 35.33, 6.75, 0, 47.92, -274.61], [9E9, 9E9, 9E9, 9E9, 9E9, 9E9]];
	VAR jointtarget SDP_2259 := [[-5.69, 35.43, 6.58, 0, 47.99, -275.69], [9E9, 9E9, 9E9, 9E9, 9E9, 9E9]];
	VAR jointtarget SDP_2260 := [[-5.72, 35.44, 6.57, 0, 47.99, -276.38], [9E9, 9E9, 9E9, 9E9, 9E9, 9E9]];
	VAR jointtarget SDP_2261 := [[-5.75, 35.44, 6.56, 0, 48, -277.74], [9E9, 9E9, 9E9, 9E9, 9E9, 9E9]];
	VAR jointtarget SDP_2262 := [[-5.79, 35.45, 6.55, 0, 48, -279.1], [9E9, 9E9, 9E9, 9E9, 9E9, 9E9]];
	VAR jointtarget SDP_2263 := [[-5.82, 35.45, 6.54, 0, 48.01, -280.46], [9E9, 9E9, 9E9, 9E9, 9E9, 9E9]];
	VAR jointtarget SDP_2264 := [[-5.85, 35.46, 6.53, 0, 48.01, -281.81], [9E9, 9E9, 9E9, 9E9, 9E9, 9E9]];
	VAR jointtarget SDP_2265 := [[-5.89, 35.47, 6.51, 0, 48.02, -283.17], [9E9, 9E9, 9E9, 9E9, 9E9, 9E9]];
	VAR jointtarget SDP_2266 := [[-5.92, 35.48, 6.5, 0, 48.02, -284.53], [9E9, 9E9, 9E9, 9E9, 9E9, 9E9]];
	VAR jointtarget SDP_2267 := [[-5.95, 35.49, 6.48, 0, 48.03, -285.88], [9E9, 9E9, 9E9, 9E9, 9E9, 9E9]];
	VAR jointtarget SDP_2268 := [[-5.98, 35.5, 6.46, 0, 48.04, -287.24], [9E9, 9E9, 9E9, 9E9, 9E9, 9E9]];
	VAR jointtarget SDP_2269 := [[-6.02, 35.51, 6.44, 0, 48.05, -288.59], [9E9, 9E9, 9E9, 9E9, 9E9, 9E9]];
	VAR jointtarget SDP_2270 := [[-6.14, 35.56, 6.36, 0, 48.08, -289.38], [9E9, 9E9, 9E9, 9E9, 9E9, 9E9]];
	VAR jointtarget SDP_2271 := [[-6.27, 35.61, 6.28, 0, 48.11, -289.51], [9E9, 9E9, 9E9, 9E9, 9E9, 9E9]];
	VAR jointtarget SDP_2272 := [[-6.4, 35.66, 6.19, 0, 48.15, -289.64], [9E9, 9E9, 9E9, 9E9, 9E9, 9E9]];
	VAR jointtarget SDP_2273 := [[-6.53, 35.71, 6.11, 0, 48.18, -289.77], [9E9, 9E9, 9E9, 9E9, 9E9, 9E9]];
	VAR jointtarget SDP_2274 := [[-6.66, 35.76, 6.02, 0, 48.22, -289.9], [9E9, 9E9, 9E9, 9E9, 9E9, 9E9]];
	VAR jointtarget SDP_2275 := [[-6.78, 35.81, 5.94, 0, 48.26, -290.02], [9E9, 9E9, 9E9, 9E9, 9E9, 9E9]];
	VAR jointtarget SDP_2276 := [[-6.91, 35.86, 5.85, 0, 48.29, -290.15], [9E9, 9E9, 9E9, 9E9, 9E9, 9E9]];
	VAR jointtarget SDP_2277 := [[-7.04, 35.91, 5.77, 0, 48.33, -290.28], [9E9, 9E9, 9E9, 9E9, 9E9, 9E9]];
	VAR jointtarget SDP_2278 := [[-7.16, 35.96, 5.68, 0, 48.36, -290.4], [9E9, 9E9, 9E9, 9E9, 9E9, 9E9]];
	VAR jointtarget SDP_2279 := [[-7.29, 36.01, 5.59, 0, 48.4, -290.53], [9E9, 9E9, 9E9, 9E9, 9E9, 9E9]];
	VAR jointtarget SDP_2280 := [[-7.55, 36.06, 5.5, 0, 48.44, -280.46], [9E9, 9E9, 9E9, 9E9, 9E9, 9E9]];
	VAR jointtarget SDP_2281 := [[-7.8, 36.01, 5.59, 0, 48.4, -260.07], [9E9, 9E9, 9E9, 9E9, 9E9, 9E9]];
	VAR jointtarget SDP_2282 := [[-8.03, 35.87, 5.83, 0, 48.3, -239.65], [9E9, 9E9, 9E9, 9E9, 9E9, 9E9]];
	VAR jointtarget SDP_2283 := [[-8.2, 35.65, 6.21, 0, 48.14, -219.17], [9E9, 9E9, 9E9, 9E9, 9E9, 9E9]];
	VAR jointtarget SDP_2284 := [[-8.28, 35.38, 6.67, 0, 47.95, -198.6], [9E9, 9E9, 9E9, 9E9, 9E9, 9E9]];
	VAR jointtarget SDP_2285 := [[-8.27, 35.09, 7.15, 0, 47.75, -177.95], [9E9, 9E9, 9E9, 9E9, 9E9, 9E9]];
	VAR jointtarget SDP_2286 := [[-8.17, 34.83, 7.6, 0, 47.57, -157.19], [9E9, 9E9, 9E9, 9E9, 9E9, 9E9]];
	VAR jointtarget SDP_2287 := [[-7.98, 34.63, 7.94, 0, 47.43, -136.36], [9E9, 9E9, 9E9, 9E9, 9E9, 9E9]];
	VAR jointtarget SDP_2288 := [[-7.74, 34.51, 8.15, 0, 47.34, -115.47], [9E9, 9E9, 9E9, 9E9, 9E9, 9E9]];
	VAR jointtarget SDP_2289 := [[-7.47, 34.49, 8.19, 0, 47.33, -94.56], [9E9, 9E9, 9E9, 9E9, 9E9, 9E9]];
	VAR jointtarget SDP_2290 := [[-7.34, 34.5, 8.16, 0, 47.34, -84.1], [9E9, 9E9, 9E9, 9E9, 9E9, 9E9]];
	VAR jointtarget SDP_2291 := [[-7.2, 34.51, 8.14, 0, 47.35, -83.96], [9E9, 9E9, 9E9, 9E9, 9E9, 9E9]];
	VAR jointtarget SDP_2292 := [[-7.06, 34.53, 8.11, 0, 47.36, -83.82], [9E9, 9E9, 9E9, 9E9, 9E9, 9E9]];
	VAR jointtarget SDP_2293 := [[-6.92, 34.54, 8.08, 0, 47.37, -83.68], [9E9, 9E9, 9E9, 9E9, 9E9, 9E9]];
	VAR jointtarget SDP_2294 := [[-6.79, 34.56, 8.06, 0, 47.39, -83.55], [9E9, 9E9, 9E9, 9E9, 9E9, 9E9]];
	VAR jointtarget SDP_2295 := [[-6.65, 34.57, 8.03, 0, 47.4, -83.41], [9E9, 9E9, 9E9, 9E9, 9E9, 9E9]];
	VAR jointtarget SDP_2296 := [[-6.51, 34.59, 8, 0, 47.41, -83.27], [9E9, 9E9, 9E9, 9E9, 9E9, 9E9]];
	VAR jointtarget SDP_2297 := [[-6.38, 34.6, 7.97, 0, 47.43, -83.14], [9E9, 9E9, 9E9, 9E9, 9E9, 9E9]];
	VAR jointtarget SDP_2298 := [[-6.24, 34.62, 7.94, 0, 47.44, -83], [9E9, 9E9, 9E9, 9E9, 9E9, 9E9]];
	VAR jointtarget SDP_2299 := [[-6.1, 34.64, 7.91, 0, 47.45, -82.86], [9E9, 9E9, 9E9, 9E9, 9E9, 9E9]];
	VAR jointtarget SDP_2300 := [[-6.07, 34.64, 7.9, 0, 47.46, -83.49], [9E9, 9E9, 9E9, 9E9, 9E9, 9E9]];
	VAR jointtarget SDP_2301 := [[-6.03, 34.64, 7.9, 0, 47.46, -84.78], [9E9, 9E9, 9E9, 9E9, 9E9, 9E9]];
	VAR jointtarget SDP_2302 := [[-6, 34.65, 7.89, 0, 47.46, -86.07], [9E9, 9E9, 9E9, 9E9, 9E9, 9E9]];
	VAR jointtarget SDP_2303 := [[-5.97, 34.65, 7.89, 0, 47.46, -87.36], [9E9, 9E9, 9E9, 9E9, 9E9, 9E9]];
	VAR jointtarget SDP_2304 := [[-5.93, 34.65, 7.89, 0, 47.46, -88.65], [9E9, 9E9, 9E9, 9E9, 9E9, 9E9]];
	VAR jointtarget SDP_2305 := [[-5.9, 34.65, 7.89, 0, 47.46, -89.94], [9E9, 9E9, 9E9, 9E9, 9E9, 9E9]];
	VAR jointtarget SDP_2306 := [[-5.86, 34.65, 7.89, 0, 47.46, -91.23], [9E9, 9E9, 9E9, 9E9, 9E9, 9E9]];
	VAR jointtarget SDP_2307 := [[-5.83, 34.65, 7.89, 0, 47.46, -92.52], [9E9, 9E9, 9E9, 9E9, 9E9, 9E9]];
	VAR jointtarget SDP_2308 := [[-5.79, 34.64, 7.9, 0, 47.46, -93.81], [9E9, 9E9, 9E9, 9E9, 9E9, 9E9]];
	VAR jointtarget SDP_2309 := [[-5.76, 34.64, 7.9, 0, 47.46, -95.1], [9E9, 9E9, 9E9, 9E9, 9E9, 9E9]];
	VAR jointtarget SDP_2310 := [[-4.6, 34.53, 8.09, 0, 47.38, -94.6], [9E9, 9E9, 9E9, 9E9, 9E9, 9E9]];
	VAR jointtarget SDP_2311 := [[-3.43, 34.44, 8.24, 0, 47.32, -93.43], [9E9, 9E9, 9E9, 9E9, 9E9, 9E9]];
	VAR jointtarget SDP_2312 := [[-2.26, 34.38, 8.34, 0, 47.28, -92.26], [9E9, 9E9, 9E9, 9E9, 9E9, 9E9]];
	VAR jointtarget SDP_2313 := [[-1.09, 34.35, 8.4, 0, 47.25, -91.09], [9E9, 9E9, 9E9, 9E9, 9E9, 9E9]];
	VAR jointtarget SDP_2314 := [[0.09, 34.33, 8.42, 0, 47.25, -89.91], [9E9, 9E9, 9E9, 9E9, 9E9, 9E9]];
	VAR jointtarget SDP_2315 := [[1.26, 34.35, 8.39, 0, 47.26, -88.74], [9E9, 9E9, 9E9, 9E9, 9E9, 9E9]];
	VAR jointtarget SDP_2316 := [[2.43, 34.39, 8.33, 0, 47.28, -87.57], [9E9, 9E9, 9E9, 9E9, 9E9, 9E9]];
	VAR jointtarget SDP_2317 := [[3.6, 34.45, 8.22, 0, 47.33, -86.4], [9E9, 9E9, 9E9, 9E9, 9E9, 9E9]];
	VAR jointtarget SDP_2318 := [[4.77, 34.54, 8.07, 0, 47.39, -85.23], [9E9, 9E9, 9E9, 9E9, 9E9, 9E9]];
	VAR jointtarget SDP_2319 := [[5.93, 34.66, 7.87, 0, 47.47, -84.07], [9E9, 9E9, 9E9, 9E9, 9E9, 9E9]];
	VAR jointtarget SDP_2320 := [[6.27, 34.73, 7.76, 0, 47.52, -79.23], [9E9, 9E9, 9E9, 9E9, 9E9, 9E9]];
	VAR jointtarget SDP_2321 := [[6.6, 34.85, 7.54, 0, 47.61, -69.9], [9E9, 9E9, 9E9, 9E9, 9E9, 9E9]];
	VAR jointtarget SDP_2322 := [[6.9, 35.03, 7.24, 0, 47.73, -60.6], [9E9, 9E9, 9E9, 9E9, 9E9, 9E9]];
	VAR jointtarget SDP_2323 := [[7.17, 35.26, 6.84, 0, 47.89, -51.33], [9E9, 9E9, 9E9, 9E9, 9E9, 9E9]];
	VAR jointtarget SDP_2324 := [[7.4, 35.53, 6.38, 0, 48.09, -42.1], [9E9, 9E9, 9E9, 9E9, 9E9, 9E9]];
	VAR jointtarget SDP_2325 := [[7.59, 35.85, 5.85, 0, 48.31, -32.91], [9E9, 9E9, 9E9, 9E9, 9E9, 9E9]];
	VAR jointtarget SDP_2326 := [[7.73, 36.19, 5.26, 0, 48.55, -23.77], [9E9, 9E9, 9E9, 9E9, 9E9, 9E9]];
	VAR jointtarget SDP_2327 := [[7.82, 36.55, 4.65, 0, 48.81, -14.68], [9E9, 9E9, 9E9, 9E9, 9E9, 9E9]];
	VAR jointtarget SDP_2328 := [[7.85, 36.92, 4.01, 0, 49.08, -5.65], [9E9, 9E9, 9E9, 9E9, 9E9, 9E9]];
	VAR jointtarget SDP_2329 := [[7.83, 37.29, 3.36, 0, 49.35, 3.33], [9E9, 9E9, 9E9, 9E9, 9E9, 9E9]];
	VAR jointtarget SDP_2330 := [[7.68, 38.55, 1.19, 0, 50.26, 7.68], [9E9, 9E9, 9E9, 9E9, 9E9, 9E9]];
	VAR jointtarget SDP_2331 := [[7.54, 39.82, -1.03, 0, 51.21, 7.54], [9E9, 9E9, 9E9, 9E9, 9E9, 9E9]];
	VAR jointtarget SDP_2332 := [[7.4, 41.11, -3.29, 0, 52.18, 7.4], [9E9, 9E9, 9E9, 9E9, 9E9, 9E9]];
	VAR jointtarget SDP_2333 := [[7.26, 42.42, -5.6, 0, 53.18, 7.26], [9E9, 9E9, 9E9, 9E9, 9E9, 9E9]];
	VAR jointtarget SDP_2334 := [[7.13, 43.76, -7.97, 0, 54.21, 7.13], [9E9, 9E9, 9E9, 9E9, 9E9, 9E9]];
	VAR jointtarget SDP_2335 := [[7.01, 45.12, -10.4, 0, 55.28, 7.01], [9E9, 9E9, 9E9, 9E9, 9E9, 9E9]];
	VAR jointtarget SDP_2336 := [[6.89, 46.51, -12.89, 0, 56.38, 6.89], [9E9, 9E9, 9E9, 9E9, 9E9, 9E9]];
	VAR jointtarget SDP_2337 := [[6.77, 47.94, -15.46, 0, 57.52, 6.77], [9E9, 9E9, 9E9, 9E9, 9E9, 9E9]];
	VAR jointtarget SDP_2338 := [[6.66, 49.41, -18.11, 0, 58.7, 6.66], [9E9, 9E9, 9E9, 9E9, 9E9, 9E9]];
	VAR jointtarget SDP_2339 := [[6.55, 50.91, -20.85, 0, 59.94, 6.55], [9E9, 9E9, 9E9, 9E9, 9E9, 9E9]];
	VAR jointtarget SDP_2340 := [[6.55, 50.96, -20.93, 0, 59.97, 5.89], [9E9, 9E9, 9E9, 9E9, 9E9, 9E9]];
	VAR jointtarget SDP_2341 := [[6.55, 51, -21.01, 0, 60.01, 4.56], [9E9, 9E9, 9E9, 9E9, 9E9, 9E9]];
	VAR jointtarget SDP_2342 := [[6.55, 51.05, -21.1, 0, 60.05, 3.24], [9E9, 9E9, 9E9, 9E9, 9E9, 9E9]];
	VAR jointtarget SDP_2343 := [[6.54, 51.1, -21.18, 0, 60.08, 1.91], [9E9, 9E9, 9E9, 9E9, 9E9, 9E9]];
	VAR jointtarget SDP_2344 := [[6.54, 51.14, -21.26, 0, 60.12, 0.59], [9E9, 9E9, 9E9, 9E9, 9E9, 9E9]];
	VAR jointtarget SDP_2345 := [[6.54, 51.19, -21.35, 0, 60.16, -0.74], [9E9, 9E9, 9E9, 9E9, 9E9, 9E9]];
	VAR jointtarget SDP_2346 := [[6.55, 51.23, -21.43, 0, 60.2, -2.06], [9E9, 9E9, 9E9, 9E9, 9E9, 9E9]];
	VAR jointtarget SDP_2347 := [[6.55, 51.28, -21.51, 0, 60.23, -3.38], [9E9, 9E9, 9E9, 9E9, 9E9, 9E9]];
	VAR jointtarget SDP_2348 := [[6.55, 51.32, -21.59, 0, 60.27, -4.7], [9E9, 9E9, 9E9, 9E9, 9E9, 9E9]];
	VAR jointtarget SDP_2349 := [[6.55, 51.37, -21.68, 0, 60.31, -6.03], [9E9, 9E9, 9E9, 9E9, 9E9, 9E9]];
	VAR jointtarget SDP_2350 := [[6.57, 51.55, -22.01, 0, 60.46, -6.68], [9E9, 9E9, 9E9, 9E9, 9E9, 9E9]];
	VAR jointtarget SDP_2351 := [[6.58, 51.73, -22.35, 0, 60.61, -6.66], [9E9, 9E9, 9E9, 9E9, 9E9, 9E9]];
	VAR jointtarget SDP_2352 := [[6.59, 51.92, -22.68, 0, 60.76, -6.65], [9E9, 9E9, 9E9, 9E9, 9E9, 9E9]];
	VAR jointtarget SDP_2353 := [[6.6, 52.1, -23.02, 0, 60.92, -6.64], [9E9, 9E9, 9E9, 9E9, 9E9, 9E9]];
	VAR jointtarget SDP_2354 := [[6.62, 52.29, -23.36, 0, 61.07, -6.62], [9E9, 9E9, 9E9, 9E9, 9E9, 9E9]];
	VAR jointtarget SDP_2355 := [[6.63, 52.48, -23.7, 0, 61.23, -6.61], [9E9, 9E9, 9E9, 9E9, 9E9, 9E9]];
	VAR jointtarget SDP_2356 := [[6.64, 52.67, -24.05, 0, 61.38, -6.6], [9E9, 9E9, 9E9, 9E9, 9E9, 9E9]];
	VAR jointtarget SDP_2357 := [[6.65, 52.85, -24.39, 0, 61.54, -6.59], [9E9, 9E9, 9E9, 9E9, 9E9, 9E9]];
	VAR jointtarget SDP_2358 := [[6.67, 53.04, -24.74, 0, 61.7, -6.57], [9E9, 9E9, 9E9, 9E9, 9E9, 9E9]];
	VAR jointtarget SDP_2359 := [[6.68, 53.23, -25.09, 0, 61.86, -6.56], [9E9, 9E9, 9E9, 9E9, 9E9, 9E9]];
	VAR jointtarget SDP_2360 := [[6.66, 53.61, -25.77, 0, 62.17, 3.75], [9E9, 9E9, 9E9, 9E9, 9E9, 9E9]];
	VAR jointtarget SDP_2361 := [[6.58, 53.95, -26.4, 0, 62.45, 24.31], [9E9, 9E9, 9E9, 9E9, 9E9, 9E9]];
	VAR jointtarget SDP_2362 := [[6.43, 54.22, -26.9, 0, 62.68, 44.81], [9E9, 9E9, 9E9, 9E9, 9E9, 9E9]];
	VAR jointtarget SDP_2363 := [[6.24, 54.38, -27.19, 0, 62.81, 65.27], [9E9, 9E9, 9E9, 9E9, 9E9, 9E9]];
	VAR jointtarget SDP_2364 := [[6.04, 54.41, -27.24, 0, 62.83, 85.71], [9E9, 9E9, 9E9, 9E9, 9E9, 9E9]];
	VAR jointtarget SDP_2365 := [[5.84, 54.3, -27.04, 0, 62.74, 106.16], [9E9, 9E9, 9E9, 9E9, 9E9, 9E9]];
	VAR jointtarget SDP_2366 := [[5.67, 54.07, -26.62, 0, 62.55, 126.64], [9E9, 9E9, 9E9, 9E9, 9E9, 9E9]];
	VAR jointtarget SDP_2367 := [[5.56, 53.75, -26.04, 0, 62.29, 147.18], [9E9, 9E9, 9E9, 9E9, 9E9, 9E9]];
	VAR jointtarget SDP_2368 := [[5.52, 53.39, -25.37, 0, 61.98, 167.78], [9E9, 9E9, 9E9, 9E9, 9E9, 9E9]];
	VAR jointtarget SDP_2369 := [[5.55, 53.02, -24.7, 0, 61.68, 188.46], [9E9, 9E9, 9E9, 9E9, 9E9, 9E9]];
	VAR jointtarget SDP_2370 := [[5.58, 52.84, -24.37, 0, 61.53, 198.82], [9E9, 9E9, 9E9, 9E9, 9E9, 9E9]];
	VAR jointtarget SDP_2371 := [[5.62, 52.66, -24.04, 0, 61.38, 198.86], [9E9, 9E9, 9E9, 9E9, 9E9, 9E9]];
	VAR jointtarget SDP_2372 := [[5.65, 52.48, -23.71, 0, 61.23, 198.89], [9E9, 9E9, 9E9, 9E9, 9E9, 9E9]];
	VAR jointtarget SDP_2373 := [[5.69, 52.3, -23.38, 0, 61.08, 198.93], [9E9, 9E9, 9E9, 9E9, 9E9, 9E9]];
	VAR jointtarget SDP_2374 := [[5.72, 52.13, -23.06, 0, 60.93, 198.96], [9E9, 9E9, 9E9, 9E9, 9E9, 9E9]];
	VAR jointtarget SDP_2375 := [[5.76, 51.95, -22.74, 0, 60.79, 199], [9E9, 9E9, 9E9, 9E9, 9E9, 9E9]];
	VAR jointtarget SDP_2376 := [[5.79, 51.77, -22.42, 0, 60.64, 199.03], [9E9, 9E9, 9E9, 9E9, 9E9, 9E9]];
	VAR jointtarget SDP_2377 := [[5.83, 51.6, -22.1, 0, 60.5, 199.07], [9E9, 9E9, 9E9, 9E9, 9E9, 9E9]];
	VAR jointtarget SDP_2378 := [[5.87, 51.42, -21.78, 0, 60.35, 199.11], [9E9, 9E9, 9E9, 9E9, 9E9, 9E9]];
	VAR jointtarget SDP_2379 := [[5.9, 51.25, -21.46, 0, 60.21, 199.14], [9E9, 9E9, 9E9, 9E9, 9E9, 9E9]];
	VAR jointtarget SDP_2380 := [[5.91, 51.21, -21.38, 0, 60.18, 198.49], [9E9, 9E9, 9E9, 9E9, 9E9, 9E9]];
	VAR jointtarget SDP_2381 := [[5.92, 51.16, -21.3, 0, 60.14, 197.17], [9E9, 9E9, 9E9, 9E9, 9E9, 9E9]];
	VAR jointtarget SDP_2382 := [[5.93, 51.12, -21.22, 0, 60.1, 195.86], [9E9, 9E9, 9E9, 9E9, 9E9, 9E9]];
	VAR jointtarget SDP_2383 := [[5.93, 51.08, -21.14, 0, 60.07, 194.54], [9E9, 9E9, 9E9, 9E9, 9E9, 9E9]];
	VAR jointtarget SDP_2384 := [[5.94, 51.03, -21.06, 0, 60.03, 193.22], [9E9, 9E9, 9E9, 9E9, 9E9, 9E9]];
	VAR jointtarget SDP_2385 := [[5.94, 50.99, -20.98, 0, 60, 191.9], [9E9, 9E9, 9E9, 9E9, 9E9, 9E9]];
	VAR jointtarget SDP_2386 := [[5.95, 50.94, -20.9, 0, 59.96, 190.58], [9E9, 9E9, 9E9, 9E9, 9E9, 9E9]];
	VAR jointtarget SDP_2387 := [[5.95, 50.9, -20.82, 0, 59.92, 189.26], [9E9, 9E9, 9E9, 9E9, 9E9, 9E9]];
	VAR jointtarget SDP_2388 := [[5.96, 50.85, -20.74, 0, 59.89, 187.94], [9E9, 9E9, 9E9, 9E9, 9E9, 9E9]];
	VAR jointtarget SDP_2389 := [[5.96, 50.81, -20.66, 0, 59.85, 186.62], [9E9, 9E9, 9E9, 9E9, 9E9, 9E9]];
	VAR jointtarget SDP_2390 := [[6.05, 49.4, -18.09, 0, 58.69, 186.05], [9E9, 9E9, 9E9, 9E9, 9E9, 9E9]];
	VAR jointtarget SDP_2391 := [[6.15, 48.02, -15.6, 0, 57.58, 186.15], [9E9, 9E9, 9E9, 9E9, 9E9, 9E9]];
	VAR jointtarget SDP_2392 := [[6.25, 46.68, -13.19, 0, 56.51, 186.25], [9E9, 9E9, 9E9, 9E9, 9E9, 9E9]];
	VAR jointtarget SDP_2393 := [[6.35, 45.37, -10.84, 0, 55.47, 186.35], [9E9, 9E9, 9E9, 9E9, 9E9, 9E9]];
	VAR jointtarget SDP_2394 := [[6.46, 44.08, -8.55, 0, 54.46, 186.46], [9E9, 9E9, 9E9, 9E9, 9E9, 9E9]];
	VAR jointtarget SDP_2395 := [[6.56, 42.83, -6.31, 0, 53.49, 186.56], [9E9, 9E9, 9E9, 9E9, 9E9, 9E9]];
	VAR jointtarget SDP_2396 := [[6.68, 41.59, -4.13, 0, 52.54, 186.68], [9E9, 9E9, 9E9, 9E9, 9E9, 9E9]];
	VAR jointtarget SDP_2397 := [[6.79, 40.37, -1.99, 0, 51.62, 186.79], [9E9, 9E9, 9E9, 9E9, 9E9, 9E9]];
	VAR jointtarget SDP_2398 := [[6.91, 39.17, 0.11, 0, 50.72, 186.91], [9E9, 9E9, 9E9, 9E9, 9E9, 9E9]];
	VAR jointtarget SDP_2399 := [[7.04, 37.98, 2.17, 0, 49.85, 187.04], [9E9, 9E9, 9E9, 9E9, 9E9, 9E9]];
	VAR jointtarget SDP_2400 := [[7.05, 37.61, 2.82, 0, 49.57, 182.55], [9E9, 9E9, 9E9, 9E9, 9E9, 9E9]];
	VAR jointtarget SDP_2401 := [[7.02, 37.23, 3.46, 0, 49.3, 173.52], [9E9, 9E9, 9E9, 9E9, 9E9, 9E9]];
	VAR jointtarget SDP_2402 := [[6.93, 36.87, 4.09, 0, 49.04, 164.43], [9E9, 9E9, 9E9, 9E9, 9E9, 9E9]];
	VAR jointtarget SDP_2403 := [[6.78, 36.53, 4.67, 0, 48.8, 155.28], [9E9, 9E9, 9E9, 9E9, 9E9, 9E9]];
	VAR jointtarget SDP_2404 := [[6.6, 36.22, 5.2, 0, 48.58, 146.1], [9E9, 9E9, 9E9, 9E9, 9E9, 9E9]];
	VAR jointtarget SDP_2405 := [[6.36, 35.95, 5.67, 0, 48.38, 136.86], [9E9, 9E9, 9E9, 9E9, 9E9, 9E9]];
	VAR jointtarget SDP_2406 := [[6.09, 35.72, 6.06, 0, 48.22, 127.59], [9E9, 9E9, 9E9, 9E9, 9E9, 9E9]];
	VAR jointtarget SDP_2407 := [[5.79, 35.55, 6.36, 0, 48.1, 118.29], [9E9, 9E9, 9E9, 9E9, 9E9, 9E9]];
	VAR jointtarget SDP_2408 := [[5.47, 35.42, 6.56, 0, 48.01, 108.97], [9E9, 9E9, 9E9, 9E9, 9E9, 9E9]];
	VAR jointtarget SDP_2409 := [[5.13, 35.36, 6.67, 0, 47.97, 99.63], [9E9, 9E9, 9E9, 9E9, 9E9, 9E9]];
	VAR jointtarget SDP_2410 := [[4.07, 35.27, 6.83, 0, 47.9, 94.07], [9E9, 9E9, 9E9, 9E9, 9E9, 9E9]];
	VAR jointtarget SDP_2411 := [[3.01, 35.2, 6.95, 0, 47.85, 93.01], [9E9, 9E9, 9E9, 9E9, 9E9, 9E9]];
	VAR jointtarget SDP_2412 := [[1.95, 35.15, 7.03, 0, 47.82, 91.95], [9E9, 9E9, 9E9, 9E9, 9E9, 9E9]];
	VAR jointtarget SDP_2413 := [[0.89, 35.12, 7.08, 0, 47.8, 90.89], [9E9, 9E9, 9E9, 9E9, 9E9, 9E9]];
	VAR jointtarget SDP_2414 := [[-0.18, 35.12, 7.09, 0, 47.79, 89.82], [9E9, 9E9, 9E9, 9E9, 9E9, 9E9]];
	VAR jointtarget SDP_2415 := [[-1.24, 35.13, 7.07, 0, 47.8, 88.76], [9E9, 9E9, 9E9, 9E9, 9E9, 9E9]];
	VAR jointtarget SDP_2416 := [[-2.31, 35.17, 7.01, 0, 47.83, 87.69], [9E9, 9E9, 9E9, 9E9, 9E9, 9E9]];
	VAR jointtarget SDP_2417 := [[-3.37, 35.22, 6.91, 0, 47.87, 86.63], [9E9, 9E9, 9E9, 9E9, 9E9, 9E9]];
	VAR jointtarget SDP_2418 := [[-4.43, 35.3, 6.78, 0, 47.92, 85.57], [9E9, 9E9, 9E9, 9E9, 9E9, 9E9]];
	VAR jointtarget SDP_2419 := [[-5.48, 35.4, 6.61, 0, 47.99, 84.52], [9E9, 9E9, 9E9, 9E9, 9E9, 9E9]];
	VAR jointtarget SDP_2420 := [[-5.59, 35.4, 6.6, 0, 48, 86.6], [9E9, 9E9, 9E9, 9E9, 9E9, 9E9]];
	VAR jointtarget SDP_2421 := [[-5.71, 35.4, 6.6, 0, 47.99, 90.88], [9E9, 9E9, 9E9, 9E9, 9E9, 9E9]];
	VAR jointtarget SDP_2422 := [[-5.82, 35.39, 6.62, 0, 47.99, 95.15], [9E9, 9E9, 9E9, 9E9, 9E9, 9E9]];
	VAR jointtarget SDP_2423 := [[-5.93, 35.37, 6.66, 0, 47.97, 99.43], [9E9, 9E9, 9E9, 9E9, 9E9, 9E9]];
	VAR jointtarget SDP_2424 := [[-6.04, 35.34, 6.7, 0, 47.95, 103.71], [9E9, 9E9, 9E9, 9E9, 9E9, 9E9]];
	VAR jointtarget SDP_2425 := [[-6.14, 35.31, 6.77, 0, 47.93, 107.99], [9E9, 9E9, 9E9, 9E9, 9E9, 9E9]];
	VAR jointtarget SDP_2426 := [[-6.25, 35.26, 6.85, 0, 47.89, 112.27], [9E9, 9E9, 9E9, 9E9, 9E9, 9E9]];
	VAR jointtarget SDP_2427 := [[-6.35, 35.21, 6.94, 0, 47.86, 116.56], [9E9, 9E9, 9E9, 9E9, 9E9, 9E9]];
	VAR jointtarget SDP_2428 := [[-6.44, 35.14, 7.04, 0, 47.81, 120.85], [9E9, 9E9, 9E9, 9E9, 9E9, 9E9]];
	VAR jointtarget SDP_2429 := [[-6.54, 35.08, 7.16, 0, 47.76, 125.15], [9E9, 9E9, 9E9, 9E9, 9E9, 9E9]];
	VAR jointtarget SDP_2430 := [[-6.59, 35.03, 7.23, 0, 47.73, 127.29], [9E9, 9E9, 9E9, 9E9, 9E9, 9E9]];
	VAR jointtarget SDP_2431 := [[-6.64, 34.99, 7.31, 0, 47.7, 127.23], [9E9, 9E9, 9E9, 9E9, 9E9, 9E9]];
	VAR jointtarget SDP_2432 := [[-6.7, 34.94, 7.38, 0, 47.67, 127.18], [9E9, 9E9, 9E9, 9E9, 9E9, 9E9]];
	VAR jointtarget SDP_2433 := [[-6.75, 34.9, 7.46, 0, 47.64, 127.12], [9E9, 9E9, 9E9, 9E9, 9E9, 9E9]];
	VAR jointtarget SDP_2434 := [[-6.81, 34.86, 7.53, 0, 47.61, 127.07], [9E9, 9E9, 9E9, 9E9, 9E9, 9E9]];
	VAR jointtarget SDP_2435 := [[-6.86, 34.81, 7.61, 0, 47.58, 127.01], [9E9, 9E9, 9E9, 9E9, 9E9, 9E9]];
	VAR jointtarget SDP_2436 := [[-6.92, 34.77, 7.68, 0, 47.55, 126.96], [9E9, 9E9, 9E9, 9E9, 9E9, 9E9]];
	VAR jointtarget SDP_2437 := [[-6.97, 34.73, 7.76, 0, 47.52, 126.91], [9E9, 9E9, 9E9, 9E9, 9E9, 9E9]];
	VAR jointtarget SDP_2438 := [[-7.03, 34.68, 7.83, 0, 47.49, 126.85], [9E9, 9E9, 9E9, 9E9, 9E9, 9E9]];
	VAR jointtarget SDP_2439 := [[-7.08, 34.64, 7.9, 0, 47.46, 126.8], [9E9, 9E9, 9E9, 9E9, 9E9, 9E9]];
	VAR jointtarget SDP_2440 := [[-7.39, 34.5, 8.14, 0, 47.36, 113.1], [9E9, 9E9, 9E9, 9E9, 9E9, 9E9]];
	VAR jointtarget SDP_2441 := [[-7.72, 34.52, 8.1, 0, 47.38, 85.99], [9E9, 9E9, 9E9, 9E9, 9E9, 9E9]];
	VAR jointtarget SDP_2442 := [[-8.01, 34.7, 7.79, 0, 47.5, 58.93], [9E9, 9E9, 9E9, 9E9, 9E9, 9E9]];
	VAR jointtarget SDP_2443 := [[-8.18, 35, 7.28, 0, 47.71, 31.98], [9E9, 9E9, 9E9, 9E9, 9E9, 9E9]];
	VAR jointtarget SDP_2444 := [[-8.21, 35.35, 6.69, 0, 47.96, 5.18], [9E9, 9E9, 9E9, 9E9, 9E9, 9E9]];
	VAR jointtarget SDP_2445 := [[-8.09, 35.68, 6.12, 0, 48.19, -21.48], [9E9, 9E9, 9E9, 9E9, 9E9, 9E9]];
	VAR jointtarget SDP_2446 := [[-7.85, 35.92, 5.72, 0, 48.36, -48.01], [9E9, 9E9, 9E9, 9E9, 9E9, 9E9]];
	VAR jointtarget SDP_2447 := [[-7.53, 36.01, 5.56, 0, 48.43, -74.47], [9E9, 9E9, 9E9, 9E9, 9E9, 9E9]];
	VAR jointtarget SDP_2448 := [[-7.21, 35.94, 5.68, 0, 48.38, -100.93], [9E9, 9E9, 9E9, 9E9, 9E9, 9E9]];
	VAR jointtarget SDP_2449 := [[-6.96, 35.73, 6.05, 0, 48.23, -127.44], [9E9, 9E9, 9E9, 9E9, 9E9, 9E9]];
	VAR jointtarget SDP_2450 := [[-6.9, 35.66, 6.17, 0, 48.17, -140.78], [9E9, 9E9, 9E9, 9E9, 9E9, 9E9]];
	VAR jointtarget SDP_2451 := [[-6.85, 35.59, 6.29, 0, 48.12, -140.72], [9E9, 9E9, 9E9, 9E9, 9E9, 9E9]];
	VAR jointtarget SDP_2452 := [[-6.79, 35.51, 6.41, 0, 48.07, -140.67], [9E9, 9E9, 9E9, 9E9, 9E9, 9E9]];
	VAR jointtarget SDP_2453 := [[-6.74, 35.44, 6.53, 0, 48.02, -140.62], [9E9, 9E9, 9E9, 9E9, 9E9, 9E9]];
	VAR jointtarget SDP_2454 := [[-6.68, 35.37, 6.66, 0, 47.97, -140.56], [9E9, 9E9, 9E9, 9E9, 9E9, 9E9]];
	VAR jointtarget SDP_2455 := [[-6.63, 35.3, 6.78, 0, 47.92, -140.51], [9E9, 9E9, 9E9, 9E9, 9E9, 9E9]];
	VAR jointtarget SDP_2456 := [[-6.58, 35.23, 6.9, 0, 47.87, -140.45], [9E9, 9E9, 9E9, 9E9, 9E9, 9E9]];
	VAR jointtarget SDP_2457 := [[-6.52, 35.16, 7.02, 0, 47.82, -140.4], [9E9, 9E9, 9E9, 9E9, 9E9, 9E9]];
	VAR jointtarget SDP_2458 := [[-6.47, 35.09, 7.14, 0, 47.77, -140.34], [9E9, 9E9, 9E9, 9E9, 9E9, 9E9]];
	VAR jointtarget SDP_2459 := [[-6.41, 35.02, 7.26, 0, 47.72, -140.29], [9E9, 9E9, 9E9, 9E9, 9E9, 9E9]];
	VAR jointtarget SDP_2460 := [[-6.38, 34.99, 7.31, 0, 47.7, -139.16], [9E9, 9E9, 9E9, 9E9, 9E9, 9E9]];
	VAR jointtarget SDP_2461 := [[-6.36, 34.95, 7.37, 0, 47.68, -136.92], [9E9, 9E9, 9E9, 9E9, 9E9, 9E9]];
	VAR jointtarget SDP_2462 := [[-6.33, 34.93, 7.41, 0, 47.66, -134.69], [9E9, 9E9, 9E9, 9E9, 9E9, 9E9]];
	VAR jointtarget SDP_2463 := [[-6.3, 34.9, 7.46, 0, 47.64, -132.45], [9E9, 9E9, 9E9, 9E9, 9E9, 9E9]];
	VAR jointtarget SDP_2464 := [[-6.27, 34.87, 7.51, 0, 47.62, -130.22], [9E9, 9E9, 9E9, 9E9, 9E9, 9E9]];
	VAR jointtarget SDP_2465 := [[-6.24, 34.84, 7.55, 0, 47.61, -127.98], [9E9, 9E9, 9E9, 9E9, 9E9, 9E9]];
	VAR jointtarget SDP_2466 := [[-6.21, 34.82, 7.59, 0, 47.59, -125.74], [9E9, 9E9, 9E9, 9E9, 9E9, 9E9]];
	VAR jointtarget SDP_2467 := [[-6.18, 34.79, 7.63, 0, 47.57, -123.5], [9E9, 9E9, 9E9, 9E9, 9E9, 9E9]];
	VAR jointtarget SDP_2468 := [[-6.14, 34.77, 7.67, 0, 47.56, -121.26], [9E9, 9E9, 9E9, 9E9, 9E9, 9E9]];
	VAR jointtarget SDP_2469 := [[-6.11, 34.75, 7.7, 0, 47.55, -119.01], [9E9, 9E9, 9E9, 9E9, 9E9, 9E9]];
	VAR jointtarget SDP_2470 := [[-6.09, 34.74, 7.72, 0, 47.54, -117.89], [9E9, 9E9, 9E9, 9E9, 9E9, 9E9]];
	VAR jointtarget SDP_2471 := [[-6.07, 34.73, 7.74, 0, 47.54, -117.87], [9E9, 9E9, 9E9, 9E9, 9E9, 9E9]];
	VAR jointtarget SDP_2472 := [[-6.05, 34.72, 7.75, 0, 47.53, -117.86], [9E9, 9E9, 9E9, 9E9, 9E9, 9E9]];
	VAR jointtarget SDP_2473 := [[-6.04, 34.71, 7.77, 0, 47.52, -117.84], [9E9, 9E9, 9E9, 9E9, 9E9, 9E9]];
	VAR jointtarget SDP_2474 := [[-6.02, 34.7, 7.79, 0, 47.52, -117.82], [9E9, 9E9, 9E9, 9E9, 9E9, 9E9]];
	VAR jointtarget SDP_2475 := [[-6, 34.69, 7.8, 0, 47.51, -117.8], [9E9, 9E9, 9E9, 9E9, 9E9, 9E9]];
	VAR jointtarget SDP_2476 := [[-5.98, 34.68, 7.82, 0, 47.51, -117.79], [9E9, 9E9, 9E9, 9E9, 9E9, 9E9]];
	VAR jointtarget SDP_2477 := [[-5.97, 34.67, 7.83, 0, 47.5, -117.77], [9E9, 9E9, 9E9, 9E9, 9E9, 9E9]];
	VAR jointtarget SDP_2478 := [[-5.95, 34.66, 7.85, 0, 47.49, -117.75], [9E9, 9E9, 9E9, 9E9, 9E9, 9E9]];
	VAR jointtarget SDP_2479 := [[-5.93, 34.64, 7.87, 0, 47.49, -117.73], [9E9, 9E9, 9E9, 9E9, 9E9, 9E9]];
	VAR jointtarget SDP_2480 := [[-4.75, 34.53, 8.07, 0, 47.41, -94.75], [9E9, 9E9, 9E9, 9E9, 9E9, 9E9]];
	VAR jointtarget SDP_2481 := [[-3.57, 34.44, 8.22, 0, 47.34, -93.57], [9E9, 9E9, 9E9, 9E9, 9E9, 9E9]];
	VAR jointtarget SDP_2482 := [[-2.38, 34.37, 8.33, 0, 47.3, -92.38], [9E9, 9E9, 9E9, 9E9, 9E9, 9E9]];
	VAR jointtarget SDP_2483 := [[-1.19, 34.33, 8.39, 0, 47.27, -91.19], [9E9, 9E9, 9E9, 9E9, 9E9, 9E9]];
	VAR jointtarget SDP_2484 := [[0, 34.32, 8.42, 0, 47.26, -90], [9E9, 9E9, 9E9, 9E9, 9E9, 9E9]];
	VAR jointtarget SDP_2485 := [[1.19, 34.33, 8.39, 0, 47.27, -88.81], [9E9, 9E9, 9E9, 9E9, 9E9, 9E9]];
	VAR jointtarget SDP_2486 := [[2.38, 34.37, 8.33, 0, 47.3, -87.62], [9E9, 9E9, 9E9, 9E9, 9E9, 9E9]];
	VAR jointtarget SDP_2487 := [[3.57, 34.44, 8.22, 0, 47.34, -86.43], [9E9, 9E9, 9E9, 9E9, 9E9, 9E9]];
	VAR jointtarget SDP_2488 := [[4.75, 34.53, 8.07, 0, 47.41, -85.25], [9E9, 9E9, 9E9, 9E9, 9E9, 9E9]];
	VAR jointtarget SDP_2489 := [[5.93, 34.64, 7.87, 0, 47.49, -84.07], [9E9, 9E9, 9E9, 9E9, 9E9, 9E9]];
	VAR jointtarget SDP_2490 := [[6.27, 34.71, 7.75, 0, 47.53, -79.23], [9E9, 9E9, 9E9, 9E9, 9E9, 9E9]];
	VAR jointtarget SDP_2491 := [[6.6, 34.84, 7.54, 0, 47.62, -69.9], [9E9, 9E9, 9E9, 9E9, 9E9, 9E9]];
	VAR jointtarget SDP_2492 := [[6.9, 35.02, 7.23, 0, 47.75, -60.6], [9E9, 9E9, 9E9, 9E9, 9E9, 9E9]];
	VAR jointtarget SDP_2493 := [[7.17, 35.25, 6.84, 0, 47.91, -51.33], [9E9, 9E9, 9E9, 9E9, 9E9, 9E9]];
	VAR jointtarget SDP_2494 := [[7.4, 35.52, 6.37, 0, 48.1, -42.1], [9E9, 9E9, 9E9, 9E9, 9E9, 9E9]];
	VAR jointtarget SDP_2495 := [[7.59, 35.83, 5.84, 0, 48.32, -32.91], [9E9, 9E9, 9E9, 9E9, 9E9, 9E9]];
	VAR jointtarget SDP_2496 := [[7.73, 36.17, 5.26, 0, 48.57, -23.77], [9E9, 9E9, 9E9, 9E9, 9E9, 9E9]];
	VAR jointtarget SDP_2497 := [[7.82, 36.53, 4.64, 0, 48.82, -14.68], [9E9, 9E9, 9E9, 9E9, 9E9, 9E9]];
	VAR jointtarget SDP_2498 := [[7.85, 36.91, 4, 0, 49.09, -5.65], [9E9, 9E9, 9E9, 9E9, 9E9, 9E9]];
	VAR jointtarget SDP_2499 := [[7.83, 37.28, 3.36, 0, 49.36, 3.33], [9E9, 9E9, 9E9, 9E9, 9E9, 9E9]];
	VAR jointtarget SDP_2500 := [[7.68, 38.51, 1.23, 0, 50.26, 7.68], [9E9, 9E9, 9E9, 9E9, 9E9, 9E9]];
	VAR jointtarget SDP_2501 := [[7.54, 39.76, -0.95, 0, 51.19, 7.54], [9E9, 9E9, 9E9, 9E9, 9E9, 9E9]];
	VAR jointtarget SDP_2502 := [[7.4, 41.03, -3.17, 0, 52.14, 7.4], [9E9, 9E9, 9E9, 9E9, 9E9, 9E9]];
	VAR jointtarget SDP_2503 := [[7.27, 42.32, -5.44, 0, 53.12, 7.27], [9E9, 9E9, 9E9, 9E9, 9E9, 9E9]];
	VAR jointtarget SDP_2504 := [[7.15, 43.63, -7.76, 0, 54.13, 7.15], [9E9, 9E9, 9E9, 9E9, 9E9, 9E9]];
	VAR jointtarget SDP_2505 := [[7.02, 44.96, -10.14, 0, 55.17, 7.02], [9E9, 9E9, 9E9, 9E9, 9E9, 9E9]];
	VAR jointtarget SDP_2506 := [[6.9, 46.33, -12.58, 0, 56.25, 6.9], [9E9, 9E9, 9E9, 9E9, 9E9, 9E9]];
	VAR jointtarget SDP_2507 := [[6.79, 47.72, -15.09, 0, 57.37, 6.79], [9E9, 9E9, 9E9, 9E9, 9E9, 9E9]];
	VAR jointtarget SDP_2508 := [[6.68, 49.16, -17.68, 0, 58.52, 6.68], [9E9, 9E9, 9E9, 9E9, 9E9, 9E9]];
	VAR jointtarget SDP_2509 := [[6.57, 50.63, -20.36, 0, 59.73, 6.57], [9E9, 9E9, 9E9, 9E9, 9E9, 9E9]];
	VAR jointtarget SDP_2510 := [[6.56, 50.78, -20.63, 0, 59.85, 8.75], [9E9, 9E9, 9E9, 9E9, 9E9, 9E9]];
	VAR jointtarget SDP_2511 := [[6.54, 50.92, -20.89, 0, 59.97, 13.12], [9E9, 9E9, 9E9, 9E9, 9E9, 9E9]];
	VAR jointtarget SDP_2512 := [[6.51, 51.07, -21.15, 0, 60.08, 17.48], [9E9, 9E9, 9E9, 9E9, 9E9, 9E9]];
	VAR jointtarget SDP_2513 := [[6.48, 51.21, -21.41, 0, 60.2, 21.83], [9E9, 9E9, 9E9, 9E9, 9E9, 9E9]];
	VAR jointtarget SDP_2514 := [[6.44, 51.34, -21.65, 0, 60.31, 26.18], [9E9, 9E9, 9E9, 9E9, 9E9, 9E9]];
	VAR jointtarget SDP_2515 := [[6.39, 51.47, -21.89, 0, 60.42, 30.52], [9E9, 9E9, 9E9, 9E9, 9E9, 9E9]];
	VAR jointtarget SDP_2516 := [[6.34, 51.6, -22.12, 0, 60.52, 34.86], [9E9, 9E9, 9E9, 9E9, 9E9, 9E9]];
	VAR jointtarget SDP_2517 := [[6.28, 51.72, -22.33, 0, 60.62, 39.19], [9E9, 9E9, 9E9, 9E9, 9E9, 9E9]];
	VAR jointtarget SDP_2518 := [[6.22, 51.83, -22.54, 0, 60.71, 43.51], [9E9, 9E9, 9E9, 9E9, 9E9, 9E9]];
	VAR jointtarget SDP_2519 := [[6.15, 51.93, -22.72, 0, 60.79, 47.83], [9E9, 9E9, 9E9, 9E9, 9E9, 9E9]];
	VAR jointtarget SDP_2520 := [[6.11, 51.99, -22.83, 0, 60.84, 49.99], [9E9, 9E9, 9E9, 9E9, 9E9, 9E9]];
	VAR jointtarget SDP_2521 := [[6.07, 52.05, -22.94, 0, 60.89, 49.95], [9E9, 9E9, 9E9, 9E9, 9E9, 9E9]];
	VAR jointtarget SDP_2522 := [[6.03, 52.11, -23.05, 0, 60.94, 49.9], [9E9, 9E9, 9E9, 9E9, 9E9, 9E9]];
	VAR jointtarget SDP_2523 := [[5.99, 52.17, -23.16, 0, 60.99, 49.86], [9E9, 9E9, 9E9, 9E9, 9E9, 9E9]];
	VAR jointtarget SDP_2524 := [[5.94, 52.23, -23.27, 0, 61.04, 49.82], [9E9, 9E9, 9E9, 9E9, 9E9, 9E9]];
	VAR jointtarget SDP_2525 := [[5.9, 52.29, -23.38, 0, 61.09, 49.78], [9E9, 9E9, 9E9, 9E9, 9E9, 9E9]];
	VAR jointtarget SDP_2526 := [[5.86, 52.35, -23.49, 0, 61.14, 49.74], [9E9, 9E9, 9E9, 9E9, 9E9, 9E9]];
	VAR jointtarget SDP_2527 := [[5.82, 52.41, -23.6, 0, 61.19, 49.7], [9E9, 9E9, 9E9, 9E9, 9E9, 9E9]];
	VAR jointtarget SDP_2528 := [[5.78, 52.47, -23.71, 0, 61.24, 49.66], [9E9, 9E9, 9E9, 9E9, 9E9, 9E9]];
	VAR jointtarget SDP_2529 := [[5.74, 52.53, -23.82, 0, 61.29, 49.61], [9E9, 9E9, 9E9, 9E9, 9E9, 9E9]];
	VAR jointtarget SDP_2530 := [[5.58, 52.9, -24.5, 0, 61.6, 36.07], [9E9, 9E9, 9E9, 9E9, 9E9, 9E9]];
	VAR jointtarget SDP_2531 := [[5.54, 53.36, -25.33, 0, 61.98, 9.25], [9E9, 9E9, 9E9, 9E9, 9E9, 9E9]];
	VAR jointtarget SDP_2532 := [[5.62, 53.8, -26.15, 0, 62.35, -17.44], [9E9, 9E9, 9E9, 9E9, 9E9, 9E9]];
	VAR jointtarget SDP_2533 := [[5.8, 54.14, -26.77, 0, 62.63, -44.04], [9E9, 9E9, 9E9, 9E9, 9E9, 9E9]];
	VAR jointtarget SDP_2534 := [[6.04, 54.3, -27.06, 0, 62.76, -70.57], [9E9, 9E9, 9E9, 9E9, 9E9, 9E9]];
	VAR jointtarget SDP_2535 := [[6.3, 54.24, -26.95, 0, 62.71, -97.09], [9E9, 9E9, 9E9, 9E9, 9E9, 9E9]];
	VAR jointtarget SDP_2536 := [[6.51, 53.97, -26.47, 0, 62.49, -123.65], [9E9, 9E9, 9E9, 9E9, 9E9, 9E9]];
	VAR jointtarget SDP_2537 := [[6.64, 53.57, -25.72, 0, 62.15, -150.3], [9E9, 9E9, 9E9, 9E9, 9E9, 9E9]];
	VAR jointtarget SDP_2538 := [[6.66, 53.1, -24.87, 0, 61.77, -177.06], [9E9, 9E9, 9E9, 9E9, 9E9, 9E9]];
	VAR jointtarget SDP_2539 := [[6.55, 52.68, -24.1, 0, 61.42, -203.94], [9E9, 9E9, 9E9, 9E9, 9E9, 9E9]];
	VAR jointtarget SDP_2540 := [[6.52, 52.61, -23.96, 0, 61.36, -217.36], [9E9, 9E9, 9E9, 9E9, 9E9, 9E9]];
	VAR jointtarget SDP_2541 := [[6.48, 52.53, -23.83, 0, 61.29, -217.39], [9E9, 9E9, 9E9, 9E9, 9E9, 9E9]];
	VAR jointtarget SDP_2542 := [[6.45, 52.46, -23.69, 0, 61.23, -217.42], [9E9, 9E9, 9E9, 9E9, 9E9, 9E9]];
	VAR jointtarget SDP_2543 := [[6.42, 52.38, -23.55, 0, 61.17, -217.46], [9E9, 9E9, 9E9, 9E9, 9E9, 9E9]];
	VAR jointtarget SDP_2544 := [[6.39, 52.31, -23.42, 0, 61.11, -217.49], [9E9, 9E9, 9E9, 9E9, 9E9, 9E9]];
	VAR jointtarget SDP_2545 := [[6.35, 52.24, -23.28, 0, 61.05, -217.52], [9E9, 9E9, 9E9, 9E9, 9E9, 9E9]];
	VAR jointtarget SDP_2546 := [[6.32, 52.16, -23.15, 0, 60.99, -217.56], [9E9, 9E9, 9E9, 9E9, 9E9, 9E9]];
	VAR jointtarget SDP_2547 := [[6.29, 52.09, -23.01, 0, 60.93, -217.59], [9E9, 9E9, 9E9, 9E9, 9E9, 9E9]];
	VAR jointtarget SDP_2548 := [[6.25, 52.01, -22.88, 0, 60.86, -217.62], [9E9, 9E9, 9E9, 9E9, 9E9, 9E9]];
	VAR jointtarget SDP_2549 := [[6.22, 51.94, -22.75, 0, 60.8, -217.66], [9E9, 9E9, 9E9, 9E9, 9E9, 9E9]];
	VAR jointtarget SDP_2550 := [[6.17, 51.82, -22.52, 0, 60.7, -215.51], [9E9, 9E9, 9E9, 9E9, 9E9, 9E9]];
	VAR jointtarget SDP_2551 := [[6.12, 51.69, -22.28, 0, 60.59, -211.17], [9E9, 9E9, 9E9, 9E9, 9E9, 9E9]];
	VAR jointtarget SDP_2552 := [[6.08, 51.55, -22.03, 0, 60.48, -206.83], [9E9, 9E9, 9E9, 9E9, 9E9, 9E9]];
	VAR jointtarget SDP_2553 := [[6.05, 51.41, -21.78, 0, 60.37, -202.47], [9E9, 9E9, 9E9, 9E9, 9E9, 9E9]];
	VAR jointtarget SDP_2554 := [[6.02, 51.27, -21.51, 0, 60.25, -198.11], [9E9, 9E9, 9E9, 9E9, 9E9, 9E9]];
	VAR jointtarget SDP_2555 := [[6, 51.12, -21.25, 0, 60.13, -193.75], [9E9, 9E9, 9E9, 9E9, 9E9, 9E9]];
	VAR jointtarget SDP_2556 := [[5.98, 50.97, -20.98, 0, 60.01, -189.38], [9E9, 9E9, 9E9, 9E9, 9E9, 9E9]];
	VAR jointtarget SDP_2557 := [[5.97, 50.82, -20.71, 0, 59.88, -185], [9E9, 9E9, 9E9, 9E9, 9E9, 9E9]];
	VAR jointtarget SDP_2558 := [[5.97, 50.67, -20.43, 0, 59.76, -180.61], [9E9, 9E9, 9E9, 9E9, 9E9, 9E9]];
	VAR jointtarget SDP_2559 := [[5.98, 50.53, -20.16, 0, 59.64, -176.22], [9E9, 9E9, 9E9, 9E9, 9E9, 9E9]];
	VAR jointtarget SDP_2560 := [[6.07, 49.15, -17.66, 0, 58.51, -173.93], [9E9, 9E9, 9E9, 9E9, 9E9, 9E9]];
	VAR jointtarget SDP_2561 := [[6.16, 47.8, -15.23, 0, 57.43, -173.84], [9E9, 9E9, 9E9, 9E9, 9E9, 9E9]];
	VAR jointtarget SDP_2562 := [[6.26, 46.49, -12.87, 0, 56.38, -173.74], [9E9, 9E9, 9E9, 9E9, 9E9, 9E9]];
	VAR jointtarget SDP_2563 := [[6.36, 45.21, -10.58, 0, 55.37, -173.64], [9E9, 9E9, 9E9, 9E9, 9E9, 9E9]];
	VAR jointtarget SDP_2564 := [[6.47, 43.95, -8.34, 0, 54.38, -173.53], [9E9, 9E9, 9E9, 9E9, 9E9, 9E9]];
	VAR jointtarget SDP_2565 := [[6.57, 42.72, -6.15, 0, 53.43, -173.43], [9E9, 9E9, 9E9, 9E9, 9E9, 9E9]];
	VAR jointtarget SDP_2566 := [[6.68, 41.51, -4.01, 0, 52.5, -173.32], [9E9, 9E9, 9E9, 9E9, 9E9, 9E9]];
	VAR jointtarget SDP_2567 := [[6.8, 40.31, -1.91, 0, 51.6, -173.2], [9E9, 9E9, 9E9, 9E9, 9E9, 9E9]];
	VAR jointtarget SDP_2568 := [[6.92, 39.13, 0.15, 0, 50.72, -173.08], [9E9, 9E9, 9E9, 9E9, 9E9, 9E9]];
	VAR jointtarget SDP_2569 := [[7.04, 37.97, 2.16, 0, 49.86, -172.96], [9E9, 9E9, 9E9, 9E9, 9E9, 9E9]];
	VAR jointtarget SDP_2570 := [[7.05, 37.59, 2.82, 0, 49.59, -177.45], [9E9, 9E9, 9E9, 9E9, 9E9, 9E9]];
	VAR jointtarget SDP_2571 := [[7.02, 37.22, 3.46, 0, 49.32, -186.48], [9E9, 9E9, 9E9, 9E9, 9E9, 9E9]];
	VAR jointtarget SDP_2572 := [[6.93, 36.86, 4.08, 0, 49.06, -195.57], [9E9, 9E9, 9E9, 9E9, 9E9, 9E9]];
	VAR jointtarget SDP_2573 := [[6.78, 36.52, 4.67, 0, 48.81, -204.72], [9E9, 9E9, 9E9, 9E9, 9E9, 9E9]];
	VAR jointtarget SDP_2574 := [[6.6, 36.21, 5.2, 0, 48.59, -213.9], [9E9, 9E9, 9E9, 9E9, 9E9, 9E9]];
	VAR jointtarget SDP_2575 := [[6.36, 35.94, 5.67, 0, 48.4, -223.14], [9E9, 9E9, 9E9, 9E9, 9E9, 9E9]];
	VAR jointtarget SDP_2576 := [[6.09, 35.71, 6.05, 0, 48.24, -232.41], [9E9, 9E9, 9E9, 9E9, 9E9, 9E9]];
	VAR jointtarget SDP_2577 := [[5.79, 35.53, 6.36, 0, 48.11, -241.71], [9E9, 9E9, 9E9, 9E9, 9E9, 9E9]];
	VAR jointtarget SDP_2578 := [[5.47, 35.41, 6.56, 0, 48.03, -251.03], [9E9, 9E9, 9E9, 9E9, 9E9, 9E9]];
	VAR jointtarget SDP_2579 := [[5.13, 35.35, 6.67, 0, 47.98, -260.37], [9E9, 9E9, 9E9, 9E9, 9E9, 9E9]];
	VAR jointtarget SDP_2580 := [[4.05, 35.26, 6.83, 0, 47.92, -265.95], [9E9, 9E9, 9E9, 9E9, 9E9, 9E9]];
	VAR jointtarget SDP_2581 := [[2.97, 35.19, 6.95, 0, 47.87, -267.03], [9E9, 9E9, 9E9, 9E9, 9E9, 9E9]];
	VAR jointtarget SDP_2582 := [[1.89, 35.14, 7.03, 0, 47.83, -268.11], [9E9, 9E9, 9E9, 9E9, 9E9, 9E9]];
	VAR jointtarget SDP_2583 := [[0.8, 35.11, 7.08, 0, 47.81, -269.2], [9E9, 9E9, 9E9, 9E9, 9E9, 9E9]];
	VAR jointtarget SDP_2584 := [[-0.28, 35.1, 7.09, 0, 47.81, -270.28], [9E9, 9E9, 9E9, 9E9, 9E9, 9E9]];
	VAR jointtarget SDP_2585 := [[-1.37, 35.12, 7.06, 0, 47.82, -271.37], [9E9, 9E9, 9E9, 9E9, 9E9, 9E9]];
	VAR jointtarget SDP_2586 := [[-2.45, 35.16, 6.99, 0, 47.85, -272.45], [9E9, 9E9, 9E9, 9E9, 9E9, 9E9]];
	VAR jointtarget SDP_2587 := [[-3.53, 35.22, 6.89, 0, 47.89, -273.53], [9E9, 9E9, 9E9, 9E9, 9E9, 9E9]];
	VAR jointtarget SDP_2588 := [[-4.61, 35.3, 6.75, 0, 47.95, -274.61], [9E9, 9E9, 9E9, 9E9, 9E9, 9E9]];
	VAR jointtarget SDP_2589 := [[-5.69, 35.41, 6.57, 0, 48.02, -275.69], [9E9, 9E9, 9E9, 9E9, 9E9, 9E9]];
	VAR jointtarget SDP_2590 := [[-5.72, 35.41, 6.57, 0, 48.02, -276.38], [9E9, 9E9, 9E9, 9E9, 9E9, 9E9]];
	VAR jointtarget SDP_2591 := [[-5.75, 35.41, 6.56, 0, 48.03, -277.74], [9E9, 9E9, 9E9, 9E9, 9E9, 9E9]];
	VAR jointtarget SDP_2592 := [[-5.79, 35.42, 6.55, 0, 48.03, -279.1], [9E9, 9E9, 9E9, 9E9, 9E9, 9E9]];
	VAR jointtarget SDP_2593 := [[-5.82, 35.43, 6.54, 0, 48.04, -280.46], [9E9, 9E9, 9E9, 9E9, 9E9, 9E9]];
	VAR jointtarget SDP_2594 := [[-5.85, 35.43, 6.52, 0, 48.04, -281.81], [9E9, 9E9, 9E9, 9E9, 9E9, 9E9]];
	VAR jointtarget SDP_2595 := [[-5.89, 35.44, 6.51, 0, 48.05, -283.17], [9E9, 9E9, 9E9, 9E9, 9E9, 9E9]];
	VAR jointtarget SDP_2596 := [[-5.92, 35.45, 6.49, 0, 48.05, -284.53], [9E9, 9E9, 9E9, 9E9, 9E9, 9E9]];
	VAR jointtarget SDP_2597 := [[-5.95, 35.46, 6.48, 0, 48.06, -285.88], [9E9, 9E9, 9E9, 9E9, 9E9, 9E9]];
	VAR jointtarget SDP_2598 := [[-5.98, 35.47, 6.46, 0, 48.07, -287.24], [9E9, 9E9, 9E9, 9E9, 9E9, 9E9]];
	VAR jointtarget SDP_2599 := [[-6.02, 35.48, 6.44, 0, 48.08, -288.59], [9E9, 9E9, 9E9, 9E9, 9E9, 9E9]];
	VAR jointtarget SDP_2600 := [[-6.14, 35.53, 6.36, 0, 48.11, -289.38], [9E9, 9E9, 9E9, 9E9, 9E9, 9E9]];
	VAR jointtarget SDP_2601 := [[-6.27, 35.58, 6.27, 0, 48.15, -289.51], [9E9, 9E9, 9E9, 9E9, 9E9, 9E9]];
	VAR jointtarget SDP_2602 := [[-6.4, 35.63, 6.19, 0, 48.18, -289.64], [9E9, 9E9, 9E9, 9E9, 9E9, 9E9]];
	VAR jointtarget SDP_2603 := [[-6.53, 35.68, 6.1, 0, 48.22, -289.77], [9E9, 9E9, 9E9, 9E9, 9E9, 9E9]];
	VAR jointtarget SDP_2604 := [[-6.66, 35.73, 6.02, 0, 48.25, -289.9], [9E9, 9E9, 9E9, 9E9, 9E9, 9E9]];
	VAR jointtarget SDP_2605 := [[-6.78, 35.78, 5.93, 0, 48.29, -290.02], [9E9, 9E9, 9E9, 9E9, 9E9, 9E9]];
	VAR jointtarget SDP_2606 := [[-6.91, 35.83, 5.85, 0, 48.32, -290.15], [9E9, 9E9, 9E9, 9E9, 9E9, 9E9]];
	VAR jointtarget SDP_2607 := [[-7.04, 35.88, 5.76, 0, 48.36, -290.28], [9E9, 9E9, 9E9, 9E9, 9E9, 9E9]];
	VAR jointtarget SDP_2608 := [[-7.16, 35.93, 5.67, 0, 48.39, -290.4], [9E9, 9E9, 9E9, 9E9, 9E9, 9E9]];
	VAR jointtarget SDP_2609 := [[-7.29, 35.98, 5.59, 0, 48.43, -290.53], [9E9, 9E9, 9E9, 9E9, 9E9, 9E9]];
	VAR jointtarget SDP_2610 := [[-7.55, 36.03, 5.5, 0, 48.47, -280.46], [9E9, 9E9, 9E9, 9E9, 9E9, 9E9]];
	VAR jointtarget SDP_2611 := [[-7.8, 35.98, 5.58, 0, 48.43, -260.07], [9E9, 9E9, 9E9, 9E9, 9E9, 9E9]];
	VAR jointtarget SDP_2612 := [[-8.03, 35.84, 5.83, 0, 48.33, -239.65], [9E9, 9E9, 9E9, 9E9, 9E9, 9E9]];
	VAR jointtarget SDP_2613 := [[-8.2, 35.62, 6.21, 0, 48.17, -219.17], [9E9, 9E9, 9E9, 9E9, 9E9, 9E9]];
	VAR jointtarget SDP_2614 := [[-8.28, 35.35, 6.67, 0, 47.98, -198.6], [9E9, 9E9, 9E9, 9E9, 9E9, 9E9]];
	VAR jointtarget SDP_2615 := [[-8.27, 35.07, 7.15, 0, 47.78, -177.95], [9E9, 9E9, 9E9, 9E9, 9E9, 9E9]];
	VAR jointtarget SDP_2616 := [[-8.17, 34.81, 7.59, 0, 47.6, -157.19], [9E9, 9E9, 9E9, 9E9, 9E9, 9E9]];
	VAR jointtarget SDP_2617 := [[-7.98, 34.6, 7.94, 0, 47.46, -136.36], [9E9, 9E9, 9E9, 9E9, 9E9, 9E9]];
	VAR jointtarget SDP_2618 := [[-7.74, 34.48, 8.14, 0, 47.37, -115.47], [9E9, 9E9, 9E9, 9E9, 9E9, 9E9]];
	VAR jointtarget SDP_2619 := [[-7.47, 34.46, 8.18, 0, 47.36, -94.56], [9E9, 9E9, 9E9, 9E9, 9E9, 9E9]];
	VAR jointtarget SDP_2620 := [[-7.34, 34.47, 8.16, 0, 47.37, -84.1], [9E9, 9E9, 9E9, 9E9, 9E9, 9E9]];
	VAR jointtarget SDP_2621 := [[-7.2, 34.49, 8.13, 0, 47.38, -83.96], [9E9, 9E9, 9E9, 9E9, 9E9, 9E9]];
	VAR jointtarget SDP_2622 := [[-7.06, 34.5, 8.11, 0, 47.39, -83.82], [9E9, 9E9, 9E9, 9E9, 9E9, 9E9]];
	VAR jointtarget SDP_2623 := [[-6.92, 34.51, 8.08, 0, 47.41, -83.68], [9E9, 9E9, 9E9, 9E9, 9E9, 9E9]];
	VAR jointtarget SDP_2624 := [[-6.79, 34.53, 8.05, 0, 47.42, -83.55], [9E9, 9E9, 9E9, 9E9, 9E9, 9E9]];
	VAR jointtarget SDP_2625 := [[-6.65, 34.55, 8.02, 0, 47.43, -83.41], [9E9, 9E9, 9E9, 9E9, 9E9, 9E9]];
	VAR jointtarget SDP_2626 := [[-6.51, 34.56, 7.99, 0, 47.44, -83.27], [9E9, 9E9, 9E9, 9E9, 9E9, 9E9]];
	VAR jointtarget SDP_2627 := [[-6.38, 34.58, 7.97, 0, 47.46, -83.14], [9E9, 9E9, 9E9, 9E9, 9E9, 9E9]];
	VAR jointtarget SDP_2628 := [[-6.24, 34.59, 7.94, 0, 47.47, -83], [9E9, 9E9, 9E9, 9E9, 9E9, 9E9]];
	VAR jointtarget SDP_2629 := [[-6.1, 34.61, 7.9, 0, 47.49, -82.86], [9E9, 9E9, 9E9, 9E9, 9E9, 9E9]];
	VAR jointtarget SDP_2630 := [[-6.07, 34.61, 7.9, 0, 47.49, -83.49], [9E9, 9E9, 9E9, 9E9, 9E9, 9E9]];
	VAR jointtarget SDP_2631 := [[-6.03, 34.62, 7.89, 0, 47.49, -84.78], [9E9, 9E9, 9E9, 9E9, 9E9, 9E9]];
	VAR jointtarget SDP_2632 := [[-6, 34.62, 7.89, 0, 47.49, -86.07], [9E9, 9E9, 9E9, 9E9, 9E9, 9E9]];
	VAR jointtarget SDP_2633 := [[-5.97, 34.62, 7.88, 0, 47.49, -87.36], [9E9, 9E9, 9E9, 9E9, 9E9, 9E9]];
	VAR jointtarget SDP_2634 := [[-5.93, 34.62, 7.88, 0, 47.5, -88.65], [9E9, 9E9, 9E9, 9E9, 9E9, 9E9]];
	VAR jointtarget SDP_2635 := [[-5.9, 34.62, 7.88, 0, 47.5, -89.94], [9E9, 9E9, 9E9, 9E9, 9E9, 9E9]];
	VAR jointtarget SDP_2636 := [[-5.86, 34.62, 7.88, 0, 47.5, -91.23], [9E9, 9E9, 9E9, 9E9, 9E9, 9E9]];
	VAR jointtarget SDP_2637 := [[-5.83, 34.62, 7.89, 0, 47.49, -92.52], [9E9, 9E9, 9E9, 9E9, 9E9, 9E9]];
	VAR jointtarget SDP_2638 := [[-5.79, 34.62, 7.89, 0, 47.49, -93.81], [9E9, 9E9, 9E9, 9E9, 9E9, 9E9]];
	VAR jointtarget SDP_2639 := [[-5.76, 34.61, 7.9, 0, 47.49, -95.1], [9E9, 9E9, 9E9, 9E9, 9E9, 9E9]];
	VAR jointtarget SDP_2640 := [[-4.6, 34.5, 8.09, 0, 47.41, -94.6], [9E9, 9E9, 9E9, 9E9, 9E9, 9E9]];
	VAR jointtarget SDP_2641 := [[-3.43, 34.42, 8.23, 0, 47.35, -93.43], [9E9, 9E9, 9E9, 9E9, 9E9, 9E9]];
	VAR jointtarget SDP_2642 := [[-2.26, 34.35, 8.33, 0, 47.31, -92.26], [9E9, 9E9, 9E9, 9E9, 9E9, 9E9]];
	VAR jointtarget SDP_2643 := [[-1.09, 34.32, 8.4, 0, 47.29, -91.09], [9E9, 9E9, 9E9, 9E9, 9E9, 9E9]];
	VAR jointtarget SDP_2644 := [[0.09, 34.31, 8.41, 0, 47.28, -89.91], [9E9, 9E9, 9E9, 9E9, 9E9, 9E9]];
	VAR jointtarget SDP_2645 := [[1.26, 34.32, 8.39, 0, 47.29, -88.74], [9E9, 9E9, 9E9, 9E9, 9E9, 9E9]];
	VAR jointtarget SDP_2646 := [[2.43, 34.36, 8.32, 0, 47.32, -87.57], [9E9, 9E9, 9E9, 9E9, 9E9, 9E9]];
	VAR jointtarget SDP_2647 := [[3.6, 34.43, 8.21, 0, 47.36, -86.4], [9E9, 9E9, 9E9, 9E9, 9E9, 9E9]];
	VAR jointtarget SDP_2648 := [[4.77, 34.52, 8.06, 0, 47.42, -85.23], [9E9, 9E9, 9E9, 9E9, 9E9, 9E9]];
	VAR jointtarget SDP_2649 := [[5.93, 34.63, 7.87, 0, 47.5, -84.07], [9E9, 9E9, 9E9, 9E9, 9E9, 9E9]];
	VAR jointtarget SDP_2650 := [[6.27, 34.7, 7.75, 0, 47.55, -79.23], [9E9, 9E9, 9E9, 9E9, 9E9, 9E9]];
	VAR jointtarget SDP_2651 := [[6.6, 34.82, 7.54, 0, 47.64, -69.9], [9E9, 9E9, 9E9, 9E9, 9E9, 9E9]];
	VAR jointtarget SDP_2652 := [[6.9, 35, 7.23, 0, 47.76, -60.6], [9E9, 9E9, 9E9, 9E9, 9E9, 9E9]];
	VAR jointtarget SDP_2653 := [[7.17, 35.23, 6.84, 0, 47.93, -51.33], [9E9, 9E9, 9E9, 9E9, 9E9, 9E9]];
	VAR jointtarget SDP_2654 := [[7.4, 35.51, 6.37, 0, 48.12, -42.1], [9E9, 9E9, 9E9, 9E9, 9E9, 9E9]];
	VAR jointtarget SDP_2655 := [[7.59, 35.82, 5.84, 0, 48.34, -32.91], [9E9, 9E9, 9E9, 9E9, 9E9, 9E9]];
	VAR jointtarget SDP_2656 := [[7.73, 36.16, 5.26, 0, 48.58, -23.77], [9E9, 9E9, 9E9, 9E9, 9E9, 9E9]];
	VAR jointtarget SDP_2657 := [[7.82, 36.52, 4.64, 0, 48.84, -14.68], [9E9, 9E9, 9E9, 9E9, 9E9, 9E9]];
	VAR jointtarget SDP_2658 := [[7.85, 36.89, 4, 0, 49.11, -5.65], [9E9, 9E9, 9E9, 9E9, 9E9, 9E9]];
	VAR jointtarget SDP_2659 := [[7.83, 37.27, 3.36, 0, 49.38, 3.33], [9E9, 9E9, 9E9, 9E9, 9E9, 9E9]];
	VAR jointtarget SDP_2660 := [[7.68, 38.52, 1.18, 0, 50.29, 7.68], [9E9, 9E9, 9E9, 9E9, 9E9, 9E9]];
	VAR jointtarget SDP_2661 := [[7.54, 39.79, -1.03, 0, 51.24, 7.54], [9E9, 9E9, 9E9, 9E9, 9E9, 9E9]];
	VAR jointtarget SDP_2662 := [[7.4, 41.09, -3.29, 0, 52.21, 7.4], [9E9, 9E9, 9E9, 9E9, 9E9, 9E9]];
	VAR jointtarget SDP_2663 := [[7.26, 42.4, -5.6, 0, 53.21, 7.26], [9E9, 9E9, 9E9, 9E9, 9E9, 9E9]];
	VAR jointtarget SDP_2664 := [[7.13, 43.73, -7.97, 0, 54.24, 7.13], [9E9, 9E9, 9E9, 9E9, 9E9, 9E9]];
	VAR jointtarget SDP_2665 := [[7.01, 45.1, -10.4, 0, 55.3, 7.01], [9E9, 9E9, 9E9, 9E9, 9E9, 9E9]];
	VAR jointtarget SDP_2666 := [[6.89, 46.49, -12.9, 0, 56.4, 6.89], [9E9, 9E9, 9E9, 9E9, 9E9, 9E9]];
	VAR jointtarget SDP_2667 := [[6.77, 47.92, -15.46, 0, 57.55, 6.77], [9E9, 9E9, 9E9, 9E9, 9E9, 9E9]];
	VAR jointtarget SDP_2668 := [[6.66, 49.38, -18.11, 0, 58.73, 6.66], [9E9, 9E9, 9E9, 9E9, 9E9, 9E9]];
	VAR jointtarget SDP_2669 := [[6.55, 50.89, -20.86, 0, 59.96, 6.55], [9E9, 9E9, 9E9, 9E9, 9E9, 9E9]];
	VAR jointtarget SDP_2670 := [[6.55, 50.94, -20.94, 0, 60, 5.89], [9E9, 9E9, 9E9, 9E9, 9E9, 9E9]];
	VAR jointtarget SDP_2671 := [[6.55, 50.98, -21.02, 0, 60.04, 4.56], [9E9, 9E9, 9E9, 9E9, 9E9, 9E9]];
	VAR jointtarget SDP_2672 := [[6.55, 51.03, -21.1, 0, 60.07, 3.24], [9E9, 9E9, 9E9, 9E9, 9E9, 9E9]];
	VAR jointtarget SDP_2673 := [[6.54, 51.07, -21.19, 0, 60.11, 1.91], [9E9, 9E9, 9E9, 9E9, 9E9, 9E9]];
	VAR jointtarget SDP_2674 := [[6.54, 51.12, -21.27, 0, 60.15, 0.59], [9E9, 9E9, 9E9, 9E9, 9E9, 9E9]];
	VAR jointtarget SDP_2675 := [[6.54, 51.17, -21.35, 0, 60.19, -0.74], [9E9, 9E9, 9E9, 9E9, 9E9, 9E9]];
	VAR jointtarget SDP_2676 := [[6.55, 51.21, -21.43, 0, 60.22, -2.06], [9E9, 9E9, 9E9, 9E9, 9E9, 9E9]];
	VAR jointtarget SDP_2677 := [[6.55, 51.26, -21.52, 0, 60.26, -3.38], [9E9, 9E9, 9E9, 9E9, 9E9, 9E9]];
	VAR jointtarget SDP_2678 := [[6.55, 51.3, -21.6, 0, 60.3, -4.7], [9E9, 9E9, 9E9, 9E9, 9E9, 9E9]];
	VAR jointtarget SDP_2679 := [[6.55, 51.35, -21.68, 0, 60.34, -6.03], [9E9, 9E9, 9E9, 9E9, 9E9, 9E9]];
	VAR jointtarget SDP_2680 := [[6.57, 51.53, -22.02, 0, 60.49, -6.68], [9E9, 9E9, 9E9, 9E9, 9E9, 9E9]];
	VAR jointtarget SDP_2681 := [[6.58, 51.71, -22.35, 0, 60.64, -6.66], [9E9, 9E9, 9E9, 9E9, 9E9, 9E9]];
	VAR jointtarget SDP_2682 := [[6.59, 51.9, -22.69, 0, 60.79, -6.65], [9E9, 9E9, 9E9, 9E9, 9E9, 9E9]];
	VAR jointtarget SDP_2683 := [[6.6, 52.08, -23.03, 0, 60.94, -6.64], [9E9, 9E9, 9E9, 9E9, 9E9, 9E9]];
	VAR jointtarget SDP_2684 := [[6.62, 52.27, -23.37, 0, 61.1, -6.62], [9E9, 9E9, 9E9, 9E9, 9E9, 9E9]];
	VAR jointtarget SDP_2685 := [[6.63, 52.46, -23.71, 0, 61.25, -6.61], [9E9, 9E9, 9E9, 9E9, 9E9, 9E9]];
	VAR jointtarget SDP_2686 := [[6.64, 52.65, -24.05, 0, 61.41, -6.6], [9E9, 9E9, 9E9, 9E9, 9E9, 9E9]];
	VAR jointtarget SDP_2687 := [[6.65, 52.83, -24.4, 0, 61.56, -6.59], [9E9, 9E9, 9E9, 9E9, 9E9, 9E9]];
	VAR jointtarget SDP_2688 := [[6.67, 53.02, -24.75, 0, 61.72, -6.57], [9E9, 9E9, 9E9, 9E9, 9E9, 9E9]];
	VAR jointtarget SDP_2689 := [[6.68, 53.21, -25.09, 0, 61.88, -6.56], [9E9, 9E9, 9E9, 9E9, 9E9, 9E9]];
	VAR jointtarget SDP_2690 := [[6.66, 53.59, -25.78, 0, 62.19, 3.75], [9E9, 9E9, 9E9, 9E9, 9E9, 9E9]];
	VAR jointtarget SDP_2691 := [[6.58, 53.93, -26.41, 0, 62.48, 24.31], [9E9, 9E9, 9E9, 9E9, 9E9, 9E9]];
	VAR jointtarget SDP_2692 := [[6.43, 54.2, -26.9, 0, 62.7, 44.81], [9E9, 9E9, 9E9, 9E9, 9E9, 9E9]];
	VAR jointtarget SDP_2693 := [[6.24, 54.36, -27.19, 0, 62.84, 65.27], [9E9, 9E9, 9E9, 9E9, 9E9, 9E9]];
	VAR jointtarget SDP_2694 := [[6.04, 54.39, -27.24, 0, 62.86, 85.71], [9E9, 9E9, 9E9, 9E9, 9E9, 9E9]];
	VAR jointtarget SDP_2695 := [[5.84, 54.28, -27.05, 0, 62.77, 106.16], [9E9, 9E9, 9E9, 9E9, 9E9, 9E9]];
	VAR jointtarget SDP_2696 := [[5.67, 54.05, -26.63, 0, 62.58, 126.64], [9E9, 9E9, 9E9, 9E9, 9E9, 9E9]];
	VAR jointtarget SDP_2697 := [[5.56, 53.73, -26.05, 0, 62.31, 147.18], [9E9, 9E9, 9E9, 9E9, 9E9, 9E9]];
	VAR jointtarget SDP_2698 := [[5.52, 53.37, -25.38, 0, 62.01, 167.78], [9E9, 9E9, 9E9, 9E9, 9E9, 9E9]];
	VAR jointtarget SDP_2699 := [[5.55, 53, -24.7, 0, 61.7, 188.46], [9E9, 9E9, 9E9, 9E9, 9E9, 9E9]];
	VAR jointtarget SDP_2700 := [[5.58, 52.82, -24.37, 0, 61.55, 198.82], [9E9, 9E9, 9E9, 9E9, 9E9, 9E9]];
	VAR jointtarget SDP_2701 := [[5.62, 52.64, -24.04, 0, 61.4, 198.86], [9E9, 9E9, 9E9, 9E9, 9E9, 9E9]];
	VAR jointtarget SDP_2702 := [[5.65, 52.46, -23.72, 0, 61.25, 198.89], [9E9, 9E9, 9E9, 9E9, 9E9, 9E9]];
	VAR jointtarget SDP_2703 := [[5.69, 52.28, -23.39, 0, 61.11, 198.93], [9E9, 9E9, 9E9, 9E9, 9E9, 9E9]];
	VAR jointtarget SDP_2704 := [[5.72, 52.1, -23.07, 0, 60.96, 198.96], [9E9, 9E9, 9E9, 9E9, 9E9, 9E9]];
	VAR jointtarget SDP_2705 := [[5.76, 51.93, -22.74, 0, 60.81, 199], [9E9, 9E9, 9E9, 9E9, 9E9, 9E9]];
	VAR jointtarget SDP_2706 := [[5.79, 51.75, -22.42, 0, 60.67, 199.03], [9E9, 9E9, 9E9, 9E9, 9E9, 9E9]];
	VAR jointtarget SDP_2707 := [[5.83, 51.58, -22.1, 0, 60.52, 199.07], [9E9, 9E9, 9E9, 9E9, 9E9, 9E9]];
	VAR jointtarget SDP_2708 := [[5.87, 51.4, -21.78, 0, 60.38, 199.11], [9E9, 9E9, 9E9, 9E9, 9E9, 9E9]];
	VAR jointtarget SDP_2709 := [[5.9, 51.23, -21.47, 0, 60.24, 199.14], [9E9, 9E9, 9E9, 9E9, 9E9, 9E9]];
	VAR jointtarget SDP_2710 := [[5.91, 51.19, -21.39, 0, 60.2, 198.49], [9E9, 9E9, 9E9, 9E9, 9E9, 9E9]];
	VAR jointtarget SDP_2711 := [[5.92, 51.14, -21.31, 0, 60.17, 197.17], [9E9, 9E9, 9E9, 9E9, 9E9, 9E9]];
	VAR jointtarget SDP_2712 := [[5.93, 51.1, -21.23, 0, 60.13, 195.86], [9E9, 9E9, 9E9, 9E9, 9E9, 9E9]];
	VAR jointtarget SDP_2713 := [[5.93, 51.05, -21.15, 0, 60.09, 194.54], [9E9, 9E9, 9E9, 9E9, 9E9, 9E9]];
	VAR jointtarget SDP_2714 := [[5.94, 51.01, -21.07, 0, 60.06, 193.22], [9E9, 9E9, 9E9, 9E9, 9E9, 9E9]];
	VAR jointtarget SDP_2715 := [[5.94, 50.97, -20.99, 0, 60.02, 191.9], [9E9, 9E9, 9E9, 9E9, 9E9, 9E9]];
	VAR jointtarget SDP_2716 := [[5.95, 50.92, -20.91, 0, 59.99, 190.58], [9E9, 9E9, 9E9, 9E9, 9E9, 9E9]];
	VAR jointtarget SDP_2717 := [[5.95, 50.88, -20.83, 0, 59.95, 189.26], [9E9, 9E9, 9E9, 9E9, 9E9, 9E9]];
	VAR jointtarget SDP_2718 := [[5.96, 50.83, -20.74, 0, 59.91, 187.94], [9E9, 9E9, 9E9, 9E9, 9E9, 9E9]];
	VAR jointtarget SDP_2719 := [[5.96, 50.79, -20.66, 0, 59.87, 186.62], [9E9, 9E9, 9E9, 9E9, 9E9, 9E9]];
	VAR jointtarget SDP_2720 := [[6.05, 49.37, -18.09, 0, 58.72, 186.05], [9E9, 9E9, 9E9, 9E9, 9E9, 9E9]];
	VAR jointtarget SDP_2721 := [[6.15, 48, -15.61, 0, 57.61, 186.15], [9E9, 9E9, 9E9, 9E9, 9E9, 9E9]];
	VAR jointtarget SDP_2722 := [[6.25, 46.66, -13.19, 0, 56.54, 186.25], [9E9, 9E9, 9E9, 9E9, 9E9, 9E9]];
	VAR jointtarget SDP_2723 := [[6.35, 45.35, -10.84, 0, 55.5, 186.35], [9E9, 9E9, 9E9, 9E9, 9E9, 9E9]];
	VAR jointtarget SDP_2724 := [[6.46, 44.06, -8.55, 0, 54.49, 186.46], [9E9, 9E9, 9E9, 9E9, 9E9, 9E9]];
	VAR jointtarget SDP_2725 := [[6.56, 42.8, -6.32, 0, 53.52, 186.56], [9E9, 9E9, 9E9, 9E9, 9E9, 9E9]];
	VAR jointtarget SDP_2726 := [[6.68, 41.56, -4.13, 0, 52.57, 186.68], [9E9, 9E9, 9E9, 9E9, 9E9, 9E9]];
	VAR jointtarget SDP_2727 := [[6.79, 40.34, -1.99, 0, 51.65, 186.79], [9E9, 9E9, 9E9, 9E9, 9E9, 9E9]];
	VAR jointtarget SDP_2728 := [[6.91, 39.14, 0.1, 0, 50.75, 186.91], [9E9, 9E9, 9E9, 9E9, 9E9, 9E9]];
	VAR jointtarget SDP_2729 := [[7.04, 37.96, 2.16, 0, 49.88, 187.04], [9E9, 9E9, 9E9, 9E9, 9E9, 9E9]];
	VAR jointtarget SDP_2730 := [[7.05, 37.58, 2.81, 0, 49.61, 182.55], [9E9, 9E9, 9E9, 9E9, 9E9, 9E9]];
	VAR jointtarget SDP_2731 := [[7.02, 37.21, 3.46, 0, 49.33, 173.52], [9E9, 9E9, 9E9, 9E9, 9E9, 9E9]];
	VAR jointtarget SDP_2732 := [[6.93, 36.84, 4.08, 0, 49.07, 164.43], [9E9, 9E9, 9E9, 9E9, 9E9, 9E9]];
	VAR jointtarget SDP_2733 := [[6.78, 36.5, 4.67, 0, 48.83, 155.28], [9E9, 9E9, 9E9, 9E9, 9E9, 9E9]];
	VAR jointtarget SDP_2734 := [[6.6, 36.2, 5.2, 0, 48.61, 146.1], [9E9, 9E9, 9E9, 9E9, 9E9, 9E9]];
	VAR jointtarget SDP_2735 := [[6.36, 35.92, 5.66, 0, 48.41, 136.86], [9E9, 9E9, 9E9, 9E9, 9E9, 9E9]];
	VAR jointtarget SDP_2736 := [[6.09, 35.7, 6.05, 0, 48.25, 127.59], [9E9, 9E9, 9E9, 9E9, 9E9, 9E9]];
	VAR jointtarget SDP_2737 := [[5.79, 35.52, 6.35, 0, 48.13, 118.29], [9E9, 9E9, 9E9, 9E9, 9E9, 9E9]];
	VAR jointtarget SDP_2738 := [[5.47, 35.4, 6.56, 0, 48.04, 108.97], [9E9, 9E9, 9E9, 9E9, 9E9, 9E9]];
	VAR jointtarget SDP_2739 := [[5.13, 35.34, 6.67, 0, 48, 99.63], [9E9, 9E9, 9E9, 9E9, 9E9, 9E9]];
	VAR jointtarget SDP_2740 := [[4.07, 35.24, 6.82, 0, 47.93, 94.07], [9E9, 9E9, 9E9, 9E9, 9E9, 9E9]];
	VAR jointtarget SDP_2741 := [[3.01, 35.17, 6.94, 0, 47.88, 93.01], [9E9, 9E9, 9E9, 9E9, 9E9, 9E9]];
	VAR jointtarget SDP_2742 := [[1.95, 35.12, 7.03, 0, 47.85, 91.95], [9E9, 9E9, 9E9, 9E9, 9E9, 9E9]];
	VAR jointtarget SDP_2743 := [[0.89, 35.1, 7.07, 0, 47.83, 90.89], [9E9, 9E9, 9E9, 9E9, 9E9, 9E9]];
	VAR jointtarget SDP_2744 := [[-0.18, 35.09, 7.09, 0, 47.82, 89.82], [9E9, 9E9, 9E9, 9E9, 9E9, 9E9]];
	VAR jointtarget SDP_2745 := [[-1.24, 35.1, 7.06, 0, 47.83, 88.76], [9E9, 9E9, 9E9, 9E9, 9E9, 9E9]];
	VAR jointtarget SDP_2746 := [[-2.31, 35.14, 7, 0, 47.86, 87.69], [9E9, 9E9, 9E9, 9E9, 9E9, 9E9]];
	VAR jointtarget SDP_2747 := [[-3.37, 35.2, 6.91, 0, 47.9, 86.63], [9E9, 9E9, 9E9, 9E9, 9E9, 9E9]];
	VAR jointtarget SDP_2748 := [[-4.43, 35.27, 6.77, 0, 47.95, 85.57], [9E9, 9E9, 9E9, 9E9, 9E9, 9E9]];
	VAR jointtarget SDP_2749 := [[-5.48, 35.37, 6.61, 0, 48.02, 84.52], [9E9, 9E9, 9E9, 9E9, 9E9, 9E9]];
	VAR jointtarget SDP_2750 := [[-5.59, 35.38, 6.59, 0, 48.03, 86.6], [9E9, 9E9, 9E9, 9E9, 9E9, 9E9]];
	VAR jointtarget SDP_2751 := [[-5.71, 35.38, 6.6, 0, 48.03, 90.88], [9E9, 9E9, 9E9, 9E9, 9E9, 9E9]];
	VAR jointtarget SDP_2752 := [[-5.82, 35.36, 6.62, 0, 48.02, 95.15], [9E9, 9E9, 9E9, 9E9, 9E9, 9E9]];
	VAR jointtarget SDP_2753 := [[-5.93, 35.35, 6.65, 0, 48, 99.43], [9E9, 9E9, 9E9, 9E9, 9E9, 9E9]];
	VAR jointtarget SDP_2754 := [[-6.04, 35.32, 6.7, 0, 47.98, 103.71], [9E9, 9E9, 9E9, 9E9, 9E9, 9E9]];
	VAR jointtarget SDP_2755 := [[-6.14, 35.28, 6.76, 0, 47.96, 107.99], [9E9, 9E9, 9E9, 9E9, 9E9, 9E9]];
	VAR jointtarget SDP_2756 := [[-6.25, 35.23, 6.84, 0, 47.93, 112.27], [9E9, 9E9, 9E9, 9E9, 9E9, 9E9]];
	VAR jointtarget SDP_2757 := [[-6.35, 35.18, 6.93, 0, 47.89, 116.56], [9E9, 9E9, 9E9, 9E9, 9E9, 9E9]];
	VAR jointtarget SDP_2758 := [[-6.44, 35.12, 7.04, 0, 47.84, 120.85], [9E9, 9E9, 9E9, 9E9, 9E9, 9E9]];
	VAR jointtarget SDP_2759 := [[-6.54, 35.05, 7.16, 0, 47.8, 125.15], [9E9, 9E9, 9E9, 9E9, 9E9, 9E9]];
	VAR jointtarget SDP_2760 := [[-6.59, 35, 7.23, 0, 47.76, 127.29], [9E9, 9E9, 9E9, 9E9, 9E9, 9E9]];
	VAR jointtarget SDP_2761 := [[-6.64, 34.96, 7.3, 0, 47.73, 127.23], [9E9, 9E9, 9E9, 9E9, 9E9, 9E9]];
	VAR jointtarget SDP_2762 := [[-6.7, 34.92, 7.38, 0, 47.7, 127.18], [9E9, 9E9, 9E9, 9E9, 9E9, 9E9]];
	VAR jointtarget SDP_2763 := [[-6.75, 34.87, 7.45, 0, 47.67, 127.12], [9E9, 9E9, 9E9, 9E9, 9E9, 9E9]];
	VAR jointtarget SDP_2764 := [[-6.81, 34.83, 7.53, 0, 47.64, 127.07], [9E9, 9E9, 9E9, 9E9, 9E9, 9E9]];
	VAR jointtarget SDP_2765 := [[-6.86, 34.79, 7.6, 0, 47.61, 127.01], [9E9, 9E9, 9E9, 9E9, 9E9, 9E9]];
	VAR jointtarget SDP_2766 := [[-6.92, 34.74, 7.68, 0, 47.58, 126.96], [9E9, 9E9, 9E9, 9E9, 9E9, 9E9]];
	VAR jointtarget SDP_2767 := [[-6.97, 34.7, 7.75, 0, 47.55, 126.91], [9E9, 9E9, 9E9, 9E9, 9E9, 9E9]];
	VAR jointtarget SDP_2768 := [[-7.03, 34.66, 7.82, 0, 47.52, 126.85], [9E9, 9E9, 9E9, 9E9, 9E9, 9E9]];
	VAR jointtarget SDP_2769 := [[-7.08, 34.61, 7.9, 0, 47.49, 126.8], [9E9, 9E9, 9E9, 9E9, 9E9, 9E9]];
	VAR jointtarget SDP_2770 := [[-7.39, 34.47, 8.13, 0, 47.39, 113.1], [9E9, 9E9, 9E9, 9E9, 9E9, 9E9]];
	VAR jointtarget SDP_2771 := [[-7.72, 34.5, 8.09, 0, 47.41, 85.99], [9E9, 9E9, 9E9, 9E9, 9E9, 9E9]];
	VAR jointtarget SDP_2772 := [[-8.01, 34.68, 7.79, 0, 47.54, 58.93], [9E9, 9E9, 9E9, 9E9, 9E9, 9E9]];
	VAR jointtarget SDP_2773 := [[-8.18, 34.98, 7.28, 0, 47.74, 31.98], [9E9, 9E9, 9E9, 9E9, 9E9, 9E9]];
	VAR jointtarget SDP_2774 := [[-8.21, 35.33, 6.68, 0, 47.99, 5.18], [9E9, 9E9, 9E9, 9E9, 9E9, 9E9]];
	VAR jointtarget SDP_2775 := [[-8.09, 35.66, 6.12, 0, 48.22, -21.48], [9E9, 9E9, 9E9, 9E9, 9E9, 9E9]];
	VAR jointtarget SDP_2776 := [[-7.85, 35.89, 5.72, 0, 48.39, -48.01], [9E9, 9E9, 9E9, 9E9, 9E9, 9E9]];
	VAR jointtarget SDP_2777 := [[-7.53, 35.99, 5.55, 0, 48.46, -74.47], [9E9, 9E9, 9E9, 9E9, 9E9, 9E9]];
	VAR jointtarget SDP_2778 := [[-7.21, 35.92, 5.67, 0, 48.41, -100.93], [9E9, 9E9, 9E9, 9E9, 9E9, 9E9]];
	VAR jointtarget SDP_2779 := [[-6.96, 35.7, 6.04, 0, 48.26, -127.44], [9E9, 9E9, 9E9, 9E9, 9E9, 9E9]];
	VAR jointtarget SDP_2780 := [[-6.9, 35.63, 6.16, 0, 48.21, -140.78], [9E9, 9E9, 9E9, 9E9, 9E9, 9E9]];
	VAR jointtarget SDP_2781 := [[-6.85, 35.56, 6.29, 0, 48.16, -140.72], [9E9, 9E9, 9E9, 9E9, 9E9, 9E9]];
	VAR jointtarget SDP_2782 := [[-6.79, 35.49, 6.41, 0, 48.1, -140.67], [9E9, 9E9, 9E9, 9E9, 9E9, 9E9]];
	VAR jointtarget SDP_2783 := [[-6.74, 35.42, 6.53, 0, 48.05, -140.62], [9E9, 9E9, 9E9, 9E9, 9E9, 9E9]];
	VAR jointtarget SDP_2784 := [[-6.68, 35.35, 6.65, 0, 48, -140.56], [9E9, 9E9, 9E9, 9E9, 9E9, 9E9]];
	VAR jointtarget SDP_2785 := [[-6.63, 35.27, 6.77, 0, 47.95, -140.51], [9E9, 9E9, 9E9, 9E9, 9E9, 9E9]];
	VAR jointtarget SDP_2786 := [[-6.58, 35.2, 6.89, 0, 47.9, -140.45], [9E9, 9E9, 9E9, 9E9, 9E9, 9E9]];
	VAR jointtarget SDP_2787 := [[-6.52, 35.13, 7.01, 0, 47.85, -140.4], [9E9, 9E9, 9E9, 9E9, 9E9, 9E9]];
	VAR jointtarget SDP_2788 := [[-6.47, 35.06, 7.13, 0, 47.8, -140.34], [9E9, 9E9, 9E9, 9E9, 9E9, 9E9]];
	VAR jointtarget SDP_2789 := [[-6.41, 34.99, 7.25, 0, 47.75, -140.29], [9E9, 9E9, 9E9, 9E9, 9E9, 9E9]];
	VAR jointtarget SDP_2790 := [[-6.38, 34.96, 7.31, 0, 47.73, -139.16], [9E9, 9E9, 9E9, 9E9, 9E9, 9E9]];
	VAR jointtarget SDP_2791 := [[-6.36, 34.93, 7.36, 0, 47.71, -136.92], [9E9, 9E9, 9E9, 9E9, 9E9, 9E9]];
	VAR jointtarget SDP_2792 := [[-6.33, 34.9, 7.41, 0, 47.69, -134.69], [9E9, 9E9, 9E9, 9E9, 9E9, 9E9]];
	VAR jointtarget SDP_2793 := [[-6.3, 34.87, 7.46, 0, 47.67, -132.45], [9E9, 9E9, 9E9, 9E9, 9E9, 9E9]];
	VAR jointtarget SDP_2794 := [[-6.27, 34.84, 7.5, 0, 47.65, -130.22], [9E9, 9E9, 9E9, 9E9, 9E9, 9E9]];
	VAR jointtarget SDP_2795 := [[-6.24, 34.82, 7.55, 0, 47.64, -127.98], [9E9, 9E9, 9E9, 9E9, 9E9, 9E9]];
	VAR jointtarget SDP_2796 := [[-6.21, 34.79, 7.59, 0, 47.62, -125.74], [9E9, 9E9, 9E9, 9E9, 9E9, 9E9]];
	VAR jointtarget SDP_2797 := [[-6.18, 34.77, 7.63, 0, 47.61, -123.5], [9E9, 9E9, 9E9, 9E9, 9E9, 9E9]];
	VAR jointtarget SDP_2798 := [[-6.14, 34.74, 7.66, 0, 47.59, -121.26], [9E9, 9E9, 9E9, 9E9, 9E9, 9E9]];
	VAR jointtarget SDP_2799 := [[-6.11, 34.72, 7.7, 0, 47.58, -119.01], [9E9, 9E9, 9E9, 9E9, 9E9, 9E9]];
	VAR jointtarget SDP_2800 := [[-6.09, 34.71, 7.71, 0, 47.57, -117.89], [9E9, 9E9, 9E9, 9E9, 9E9, 9E9]];
	VAR jointtarget SDP_2801 := [[-6.07, 34.7, 7.73, 0, 47.57, -117.87], [9E9, 9E9, 9E9, 9E9, 9E9, 9E9]];
	VAR jointtarget SDP_2802 := [[-6.05, 34.69, 7.75, 0, 47.56, -117.86], [9E9, 9E9, 9E9, 9E9, 9E9, 9E9]];
	VAR jointtarget SDP_2803 := [[-6.04, 34.68, 7.76, 0, 47.56, -117.84], [9E9, 9E9, 9E9, 9E9, 9E9, 9E9]];
	VAR jointtarget SDP_2804 := [[-6.02, 34.67, 7.78, 0, 47.55, -117.82], [9E9, 9E9, 9E9, 9E9, 9E9, 9E9]];
	VAR jointtarget SDP_2805 := [[-6, 34.66, 7.8, 0, 47.54, -117.8], [9E9, 9E9, 9E9, 9E9, 9E9, 9E9]];
	VAR jointtarget SDP_2806 := [[-5.98, 34.65, 7.81, 0, 47.54, -117.79], [9E9, 9E9, 9E9, 9E9, 9E9, 9E9]];
	VAR jointtarget SDP_2807 := [[-5.97, 34.64, 7.83, 0, 47.53, -117.77], [9E9, 9E9, 9E9, 9E9, 9E9, 9E9]];
	VAR jointtarget SDP_2808 := [[-5.95, 34.63, 7.85, 0, 47.53, -117.75], [9E9, 9E9, 9E9, 9E9, 9E9, 9E9]];
	VAR jointtarget SDP_2809 := [[-5.93, 34.62, 7.86, 0, 47.52, -117.73], [9E9, 9E9, 9E9, 9E9, 9E9, 9E9]];
	VAR jointtarget SDP_2810 := [[-4.75, 34.5, 8.06, 0, 47.44, -94.75], [9E9, 9E9, 9E9, 9E9, 9E9, 9E9]];
	VAR jointtarget SDP_2811 := [[-3.57, 34.41, 8.21, 0, 47.37, -93.57], [9E9, 9E9, 9E9, 9E9, 9E9, 9E9]];
	VAR jointtarget SDP_2812 := [[-2.38, 34.35, 8.32, 0, 47.33, -92.38], [9E9, 9E9, 9E9, 9E9, 9E9, 9E9]];
	VAR jointtarget SDP_2813 := [[-1.19, 34.31, 8.39, 0, 47.3, -91.19], [9E9, 9E9, 9E9, 9E9, 9E9, 9E9]];
	VAR jointtarget SDP_2814 := [[0, 34.29, 8.41, 0, 47.29, -90], [9E9, 9E9, 9E9, 9E9, 9E9, 9E9]];
	VAR jointtarget SDP_2815 := [[1.19, 34.31, 8.39, 0, 47.3, -88.81], [9E9, 9E9, 9E9, 9E9, 9E9, 9E9]];
	VAR jointtarget SDP_2816 := [[2.38, 34.35, 8.32, 0, 47.33, -87.62], [9E9, 9E9, 9E9, 9E9, 9E9, 9E9]];
	VAR jointtarget SDP_2817 := [[3.57, 34.41, 8.21, 0, 47.37, -86.43], [9E9, 9E9, 9E9, 9E9, 9E9, 9E9]];
	VAR jointtarget SDP_2818 := [[4.75, 34.5, 8.06, 0, 47.44, -85.25], [9E9, 9E9, 9E9, 9E9, 9E9, 9E9]];
	VAR jointtarget SDP_2819 := [[5.93, 34.62, 7.86, 0, 47.52, -84.07], [9E9, 9E9, 9E9, 9E9, 9E9, 9E9]];
	VAR jointtarget SDP_2820 := [[6.27, 34.69, 7.75, 0, 47.57, -79.23], [9E9, 9E9, 9E9, 9E9, 9E9, 9E9]];
	VAR jointtarget SDP_2821 := [[6.6, 34.81, 7.53, 0, 47.65, -69.9], [9E9, 9E9, 9E9, 9E9, 9E9, 9E9]];
	VAR jointtarget SDP_2822 := [[6.9, 34.99, 7.23, 0, 47.78, -60.6], [9E9, 9E9, 9E9, 9E9, 9E9, 9E9]];
	VAR jointtarget SDP_2823 := [[7.17, 35.22, 6.84, 0, 47.94, -51.33], [9E9, 9E9, 9E9, 9E9, 9E9, 9E9]];
	VAR jointtarget SDP_2824 := [[7.4, 35.5, 6.37, 0, 48.14, -42.1], [9E9, 9E9, 9E9, 9E9, 9E9, 9E9]];
	VAR jointtarget SDP_2825 := [[7.59, 35.81, 5.84, 0, 48.36, -32.91], [9E9, 9E9, 9E9, 9E9, 9E9, 9E9]];
	VAR jointtarget SDP_2826 := [[7.73, 36.15, 5.26, 0, 48.6, -23.77], [9E9, 9E9, 9E9, 9E9, 9E9, 9E9]];
	VAR jointtarget SDP_2827 := [[7.82, 36.51, 4.64, 0, 48.85, -14.68], [9E9, 9E9, 9E9, 9E9, 9E9, 9E9]];
	VAR jointtarget SDP_2828 := [[7.85, 36.88, 4, 0, 49.12, -5.65], [9E9, 9E9, 9E9, 9E9, 9E9, 9E9]];
	VAR jointtarget SDP_2829 := [[7.83, 37.25, 3.35, 0, 49.39, 3.33], [9E9, 9E9, 9E9, 9E9, 9E9, 9E9]];
	VAR jointtarget SDP_2830 := [[7.68, 38.49, 1.22, 0, 50.29, 7.68], [9E9, 9E9, 9E9, 9E9, 9E9, 9E9]];
	VAR jointtarget SDP_2831 := [[7.54, 39.74, -0.95, 0, 51.22, 7.54], [9E9, 9E9, 9E9, 9E9, 9E9, 9E9]];
	VAR jointtarget SDP_2832 := [[7.4, 41, -3.17, 0, 52.17, 7.4], [9E9, 9E9, 9E9, 9E9, 9E9, 9E9]];
	VAR jointtarget SDP_2833 := [[7.27, 42.29, -5.44, 0, 53.15, 7.27], [9E9, 9E9, 9E9, 9E9, 9E9, 9E9]];
	VAR jointtarget SDP_2834 := [[7.15, 43.6, -7.76, 0, 54.16, 7.15], [9E9, 9E9, 9E9, 9E9, 9E9, 9E9]];
	VAR jointtarget SDP_2835 := [[7.02, 44.94, -10.14, 0, 55.2, 7.02], [9E9, 9E9, 9E9, 9E9, 9E9, 9E9]];
	VAR jointtarget SDP_2836 := [[6.9, 46.3, -12.58, 0, 56.28, 6.9], [9E9, 9E9, 9E9, 9E9, 9E9, 9E9]];
	VAR jointtarget SDP_2837 := [[6.79, 47.7, -15.1, 0, 57.39, 6.79], [9E9, 9E9, 9E9, 9E9, 9E9, 9E9]];
	VAR jointtarget SDP_2838 := [[6.68, 49.14, -17.69, 0, 58.55, 6.68], [9E9, 9E9, 9E9, 9E9, 9E9, 9E9]];
	VAR jointtarget SDP_2839 := [[6.57, 50.61, -20.36, 0, 59.75, 6.57], [9E9, 9E9, 9E9, 9E9, 9E9, 9E9]];
	VAR jointtarget SDP_2840 := [[6.56, 50.76, -20.63, 0, 59.87, 8.75], [9E9, 9E9, 9E9, 9E9, 9E9, 9E9]];
	VAR jointtarget SDP_2841 := [[6.54, 50.9, -20.9, 0, 59.99, 13.12], [9E9, 9E9, 9E9, 9E9, 9E9, 9E9]];
	VAR jointtarget SDP_2842 := [[6.51, 51.05, -21.16, 0, 60.11, 17.48], [9E9, 9E9, 9E9, 9E9, 9E9, 9E9]];
	VAR jointtarget SDP_2843 := [[6.48, 51.19, -21.41, 0, 60.22, 21.83], [9E9, 9E9, 9E9, 9E9, 9E9, 9E9]];
	VAR jointtarget SDP_2844 := [[6.44, 51.32, -21.66, 0, 60.34, 26.18], [9E9, 9E9, 9E9, 9E9, 9E9, 9E9]];
	VAR jointtarget SDP_2845 := [[6.39, 51.45, -21.9, 0, 60.44, 30.52], [9E9, 9E9, 9E9, 9E9, 9E9, 9E9]];
	VAR jointtarget SDP_2846 := [[6.34, 51.58, -22.12, 0, 60.55, 34.86], [9E9, 9E9, 9E9, 9E9, 9E9, 9E9]];
	VAR jointtarget SDP_2847 := [[6.28, 51.7, -22.34, 0, 60.64, 39.19], [9E9, 9E9, 9E9, 9E9, 9E9, 9E9]];
	VAR jointtarget SDP_2848 := [[6.22, 51.81, -22.54, 0, 60.73, 43.51], [9E9, 9E9, 9E9, 9E9, 9E9, 9E9]];
	VAR jointtarget SDP_2849 := [[6.15, 51.91, -22.73, 0, 60.82, 47.83], [9E9, 9E9, 9E9, 9E9, 9E9, 9E9]];
	VAR jointtarget SDP_2850 := [[6.11, 51.97, -22.84, 0, 60.87, 49.99], [9E9, 9E9, 9E9, 9E9, 9E9, 9E9]];
	VAR jointtarget SDP_2851 := [[6.07, 52.03, -22.95, 0, 60.92, 49.95], [9E9, 9E9, 9E9, 9E9, 9E9, 9E9]];
	VAR jointtarget SDP_2852 := [[6.03, 52.09, -23.05, 0, 60.97, 49.9], [9E9, 9E9, 9E9, 9E9, 9E9, 9E9]];
	VAR jointtarget SDP_2853 := [[5.99, 52.15, -23.16, 0, 61.02, 49.86], [9E9, 9E9, 9E9, 9E9, 9E9, 9E9]];
	VAR jointtarget SDP_2854 := [[5.94, 52.21, -23.27, 0, 61.07, 49.82], [9E9, 9E9, 9E9, 9E9, 9E9, 9E9]];
	VAR jointtarget SDP_2855 := [[5.9, 52.27, -23.38, 0, 61.12, 49.78], [9E9, 9E9, 9E9, 9E9, 9E9, 9E9]];
	VAR jointtarget SDP_2856 := [[5.86, 52.33, -23.49, 0, 61.17, 49.74], [9E9, 9E9, 9E9, 9E9, 9E9, 9E9]];
	VAR jointtarget SDP_2857 := [[5.82, 52.39, -23.61, 0, 61.22, 49.7], [9E9, 9E9, 9E9, 9E9, 9E9, 9E9]];
	VAR jointtarget SDP_2858 := [[5.78, 52.45, -23.72, 0, 61.27, 49.66], [9E9, 9E9, 9E9, 9E9, 9E9, 9E9]];
	VAR jointtarget SDP_2859 := [[5.74, 52.51, -23.83, 0, 61.32, 49.61], [9E9, 9E9, 9E9, 9E9, 9E9, 9E9]];
	VAR jointtarget SDP_2860 := [[5.58, 52.88, -24.5, 0, 61.62, 36.07], [9E9, 9E9, 9E9, 9E9, 9E9, 9E9]];
	VAR jointtarget SDP_2861 := [[5.54, 53.34, -25.34, 0, 62, 9.25], [9E9, 9E9, 9E9, 9E9, 9E9, 9E9]];
	VAR jointtarget SDP_2862 := [[5.62, 53.78, -26.16, 0, 62.38, -17.44], [9E9, 9E9, 9E9, 9E9, 9E9, 9E9]];
	VAR jointtarget SDP_2863 := [[5.8, 54.12, -26.78, 0, 62.66, -44.04], [9E9, 9E9, 9E9, 9E9, 9E9, 9E9]];
	VAR jointtarget SDP_2864 := [[6.04, 54.28, -27.07, 0, 62.79, -70.57], [9E9, 9E9, 9E9, 9E9, 9E9, 9E9]];
	VAR jointtarget SDP_2865 := [[6.3, 54.22, -26.96, 0, 62.74, -97.09], [9E9, 9E9, 9E9, 9E9, 9E9, 9E9]];
	VAR jointtarget SDP_2866 := [[6.51, 53.95, -26.47, 0, 62.52, -123.65], [9E9, 9E9, 9E9, 9E9, 9E9, 9E9]];
	VAR jointtarget SDP_2867 := [[6.64, 53.55, -25.73, 0, 62.18, -150.3], [9E9, 9E9, 9E9, 9E9, 9E9, 9E9]];
	VAR jointtarget SDP_2868 := [[6.66, 53.08, -24.88, 0, 61.79, -177.06], [9E9, 9E9, 9E9, 9E9, 9E9, 9E9]];
	VAR jointtarget SDP_2869 := [[6.55, 52.66, -24.11, 0, 61.44, -203.94], [9E9, 9E9, 9E9, 9E9, 9E9, 9E9]];
	VAR jointtarget SDP_2870 := [[6.52, 52.59, -23.97, 0, 61.38, -217.36], [9E9, 9E9, 9E9, 9E9, 9E9, 9E9]];
	VAR jointtarget SDP_2871 := [[6.48, 52.51, -23.83, 0, 61.32, -217.39], [9E9, 9E9, 9E9, 9E9, 9E9, 9E9]];
	VAR jointtarget SDP_2872 := [[6.45, 52.44, -23.7, 0, 61.26, -217.42], [9E9, 9E9, 9E9, 9E9, 9E9, 9E9]];
	VAR jointtarget SDP_2873 := [[6.42, 52.36, -23.56, 0, 61.2, -217.46], [9E9, 9E9, 9E9, 9E9, 9E9, 9E9]];
	VAR jointtarget SDP_2874 := [[6.39, 52.29, -23.42, 0, 61.13, -217.49], [9E9, 9E9, 9E9, 9E9, 9E9, 9E9]];
	VAR jointtarget SDP_2875 := [[6.35, 52.22, -23.29, 0, 61.07, -217.52], [9E9, 9E9, 9E9, 9E9, 9E9, 9E9]];
	VAR jointtarget SDP_2876 := [[6.32, 52.14, -23.15, 0, 61.01, -217.56], [9E9, 9E9, 9E9, 9E9, 9E9, 9E9]];
	VAR jointtarget SDP_2877 := [[6.29, 52.07, -23.02, 0, 60.95, -217.59], [9E9, 9E9, 9E9, 9E9, 9E9, 9E9]];
	VAR jointtarget SDP_2878 := [[6.25, 51.99, -22.88, 0, 60.89, -217.62], [9E9, 9E9, 9E9, 9E9, 9E9, 9E9]];
	VAR jointtarget SDP_2879 := [[6.22, 51.92, -22.75, 0, 60.83, -217.66], [9E9, 9E9, 9E9, 9E9, 9E9, 9E9]];
	VAR jointtarget SDP_2880 := [[6.17, 51.8, -22.52, 0, 60.73, -215.51], [9E9, 9E9, 9E9, 9E9, 9E9, 9E9]];
	VAR jointtarget SDP_2881 := [[6.12, 51.67, -22.28, 0, 60.62, -211.17], [9E9, 9E9, 9E9, 9E9, 9E9, 9E9]];
	VAR jointtarget SDP_2882 := [[6.08, 51.53, -22.04, 0, 60.51, -206.83], [9E9, 9E9, 9E9, 9E9, 9E9, 9E9]];
	VAR jointtarget SDP_2883 := [[6.05, 51.39, -21.78, 0, 60.39, -202.47], [9E9, 9E9, 9E9, 9E9, 9E9, 9E9]];
	VAR jointtarget SDP_2884 := [[6.02, 51.25, -21.52, 0, 60.27, -198.11], [9E9, 9E9, 9E9, 9E9, 9E9, 9E9]];
	VAR jointtarget SDP_2885 := [[6, 51.1, -21.25, 0, 60.15, -193.75], [9E9, 9E9, 9E9, 9E9, 9E9, 9E9]];
	VAR jointtarget SDP_2886 := [[5.98, 50.95, -20.98, 0, 60.03, -189.38], [9E9, 9E9, 9E9, 9E9, 9E9, 9E9]];
	VAR jointtarget SDP_2887 := [[5.97, 50.8, -20.71, 0, 59.91, -185], [9E9, 9E9, 9E9, 9E9, 9E9, 9E9]];
	VAR jointtarget SDP_2888 := [[5.97, 50.65, -20.44, 0, 59.79, -180.61], [9E9, 9E9, 9E9, 9E9, 9E9, 9E9]];
	VAR jointtarget SDP_2889 := [[5.98, 50.5, -20.17, 0, 59.66, -176.22], [9E9, 9E9, 9E9, 9E9, 9E9, 9E9]];
	VAR jointtarget SDP_2890 := [[6.07, 49.12, -17.67, 0, 58.54, -173.93], [9E9, 9E9, 9E9, 9E9, 9E9, 9E9]];
	VAR jointtarget SDP_2891 := [[6.16, 47.78, -15.24, 0, 57.46, -173.84], [9E9, 9E9, 9E9, 9E9, 9E9, 9E9]];
	VAR jointtarget SDP_2892 := [[6.26, 46.47, -12.88, 0, 56.41, -173.74], [9E9, 9E9, 9E9, 9E9, 9E9, 9E9]];
	VAR jointtarget SDP_2893 := [[6.36, 45.19, -10.58, 0, 55.39, -173.64], [9E9, 9E9, 9E9, 9E9, 9E9, 9E9]];
	VAR jointtarget SDP_2894 := [[6.47, 43.93, -8.34, 0, 54.41, -173.53], [9E9, 9E9, 9E9, 9E9, 9E9, 9E9]];
	VAR jointtarget SDP_2895 := [[6.57, 42.69, -6.15, 0, 53.46, -173.43], [9E9, 9E9, 9E9, 9E9, 9E9, 9E9]];
	VAR jointtarget SDP_2896 := [[6.68, 41.48, -4.01, 0, 52.53, -173.32], [9E9, 9E9, 9E9, 9E9, 9E9, 9E9]];
	VAR jointtarget SDP_2897 := [[6.8, 40.29, -1.91, 0, 51.63, -173.2], [9E9, 9E9, 9E9, 9E9, 9E9, 9E9]];
	VAR jointtarget SDP_2898 := [[6.92, 39.11, 0.14, 0, 50.75, -173.08], [9E9, 9E9, 9E9, 9E9, 9E9, 9E9]];
	VAR jointtarget SDP_2899 := [[7.04, 37.94, 2.16, 0, 49.9, -172.96], [9E9, 9E9, 9E9, 9E9, 9E9, 9E9]];
	VAR jointtarget SDP_2900 := [[7.05, 37.57, 2.81, 0, 49.62, -177.45], [9E9, 9E9, 9E9, 9E9, 9E9, 9E9]];
	VAR jointtarget SDP_2901 := [[7.02, 37.19, 3.46, 0, 49.35, -186.48], [9E9, 9E9, 9E9, 9E9, 9E9, 9E9]];
	VAR jointtarget SDP_2902 := [[6.93, 36.83, 4.08, 0, 49.09, -195.57], [9E9, 9E9, 9E9, 9E9, 9E9, 9E9]];
	VAR jointtarget SDP_2903 := [[6.78, 36.49, 4.66, 0, 48.84, -204.72], [9E9, 9E9, 9E9, 9E9, 9E9, 9E9]];
	VAR jointtarget SDP_2904 := [[6.6, 36.18, 5.2, 0, 48.62, -213.9], [9E9, 9E9, 9E9, 9E9, 9E9, 9E9]];
	VAR jointtarget SDP_2905 := [[6.36, 35.91, 5.66, 0, 48.43, -223.14], [9E9, 9E9, 9E9, 9E9, 9E9, 9E9]];
	VAR jointtarget SDP_2906 := [[6.09, 35.68, 6.05, 0, 48.27, -232.41], [9E9, 9E9, 9E9, 9E9, 9E9, 9E9]];
	VAR jointtarget SDP_2907 := [[5.79, 35.51, 6.35, 0, 48.14, -241.71], [9E9, 9E9, 9E9, 9E9, 9E9, 9E9]];
	VAR jointtarget SDP_2908 := [[5.47, 35.39, 6.56, 0, 48.06, -251.03], [9E9, 9E9, 9E9, 9E9, 9E9, 9E9]];
	VAR jointtarget SDP_2909 := [[5.13, 35.32, 6.66, 0, 48.01, -260.37], [9E9, 9E9, 9E9, 9E9, 9E9, 9E9]];
	VAR jointtarget SDP_2910 := [[4.05, 35.23, 6.82, 0, 47.95, -265.95], [9E9, 9E9, 9E9, 9E9, 9E9, 9E9]];
	VAR jointtarget SDP_2911 := [[2.97, 35.16, 6.94, 0, 47.9, -267.03], [9E9, 9E9, 9E9, 9E9, 9E9, 9E9]];
	VAR jointtarget SDP_2912 := [[1.89, 35.11, 7.03, 0, 47.86, -268.11], [9E9, 9E9, 9E9, 9E9, 9E9, 9E9]];
	VAR jointtarget SDP_2913 := [[0.8, 35.08, 7.07, 0, 47.84, -269.2], [9E9, 9E9, 9E9, 9E9, 9E9, 9E9]];
	VAR jointtarget SDP_2914 := [[-0.28, 35.08, 7.08, 0, 47.84, -270.28], [9E9, 9E9, 9E9, 9E9, 9E9, 9E9]];
	VAR jointtarget SDP_2915 := [[-1.37, 35.09, 7.05, 0, 47.85, -271.37], [9E9, 9E9, 9E9, 9E9, 9E9, 9E9]];
	VAR jointtarget SDP_2916 := [[-2.45, 35.13, 6.99, 0, 47.88, -272.45], [9E9, 9E9, 9E9, 9E9, 9E9, 9E9]];
	VAR jointtarget SDP_2917 := [[-3.53, 35.19, 6.89, 0, 47.92, -273.53], [9E9, 9E9, 9E9, 9E9, 9E9, 9E9]];
	VAR jointtarget SDP_2918 := [[-4.61, 35.27, 6.75, 0, 47.98, -274.61], [9E9, 9E9, 9E9, 9E9, 9E9, 9E9]];
	VAR jointtarget SDP_2919 := [[-5.69, 35.38, 6.57, 0, 48.05, -275.69], [9E9, 9E9, 9E9, 9E9, 9E9, 9E9]];
	VAR jointtarget SDP_2920 := [[-5.72, 35.38, 6.56, 0, 48.06, -276.38], [9E9, 9E9, 9E9, 9E9, 9E9, 9E9]];
	VAR jointtarget SDP_2921 := [[-5.75, 35.39, 6.55, 0, 48.06, -277.74], [9E9, 9E9, 9E9, 9E9, 9E9, 9E9]];
	VAR jointtarget SDP_2922 := [[-5.79, 35.39, 6.54, 0, 48.06, -279.1], [9E9, 9E9, 9E9, 9E9, 9E9, 9E9]];
	VAR jointtarget SDP_2923 := [[-5.82, 35.4, 6.53, 0, 48.07, -280.46], [9E9, 9E9, 9E9, 9E9, 9E9, 9E9]];
	VAR jointtarget SDP_2924 := [[-5.85, 35.41, 6.52, 0, 48.07, -281.81], [9E9, 9E9, 9E9, 9E9, 9E9, 9E9]];
	VAR jointtarget SDP_2925 := [[-5.89, 35.42, 6.5, 0, 48.08, -283.17], [9E9, 9E9, 9E9, 9E9, 9E9, 9E9]];
	VAR jointtarget SDP_2926 := [[-5.92, 35.43, 6.49, 0, 48.09, -284.53], [9E9, 9E9, 9E9, 9E9, 9E9, 9E9]];
	VAR jointtarget SDP_2927 := [[-5.95, 35.44, 6.47, 0, 48.09, -285.88], [9E9, 9E9, 9E9, 9E9, 9E9, 9E9]];
	VAR jointtarget SDP_2928 := [[-5.98, 35.45, 6.45, 0, 48.1, -287.24], [9E9, 9E9, 9E9, 9E9, 9E9, 9E9]];
	VAR jointtarget SDP_2929 := [[-6.02, 35.46, 6.43, 0, 48.11, -288.59], [9E9, 9E9, 9E9, 9E9, 9E9, 9E9]];
	VAR jointtarget SDP_2930 := [[-6.14, 35.51, 6.35, 0, 48.14, -289.38], [9E9, 9E9, 9E9, 9E9, 9E9, 9E9]];
	VAR jointtarget SDP_2931 := [[-6.27, 35.55, 6.27, 0, 48.18, -289.51], [9E9, 9E9, 9E9, 9E9, 9E9, 9E9]];
	VAR jointtarget SDP_2932 := [[-6.4, 35.6, 6.18, 0, 48.21, -289.64], [9E9, 9E9, 9E9, 9E9, 9E9, 9E9]];
	VAR jointtarget SDP_2933 := [[-6.53, 35.65, 6.1, 0, 48.25, -289.77], [9E9, 9E9, 9E9, 9E9, 9E9, 9E9]];
	VAR jointtarget SDP_2934 := [[-6.66, 35.7, 6.01, 0, 48.28, -289.9], [9E9, 9E9, 9E9, 9E9, 9E9, 9E9]];
